*)
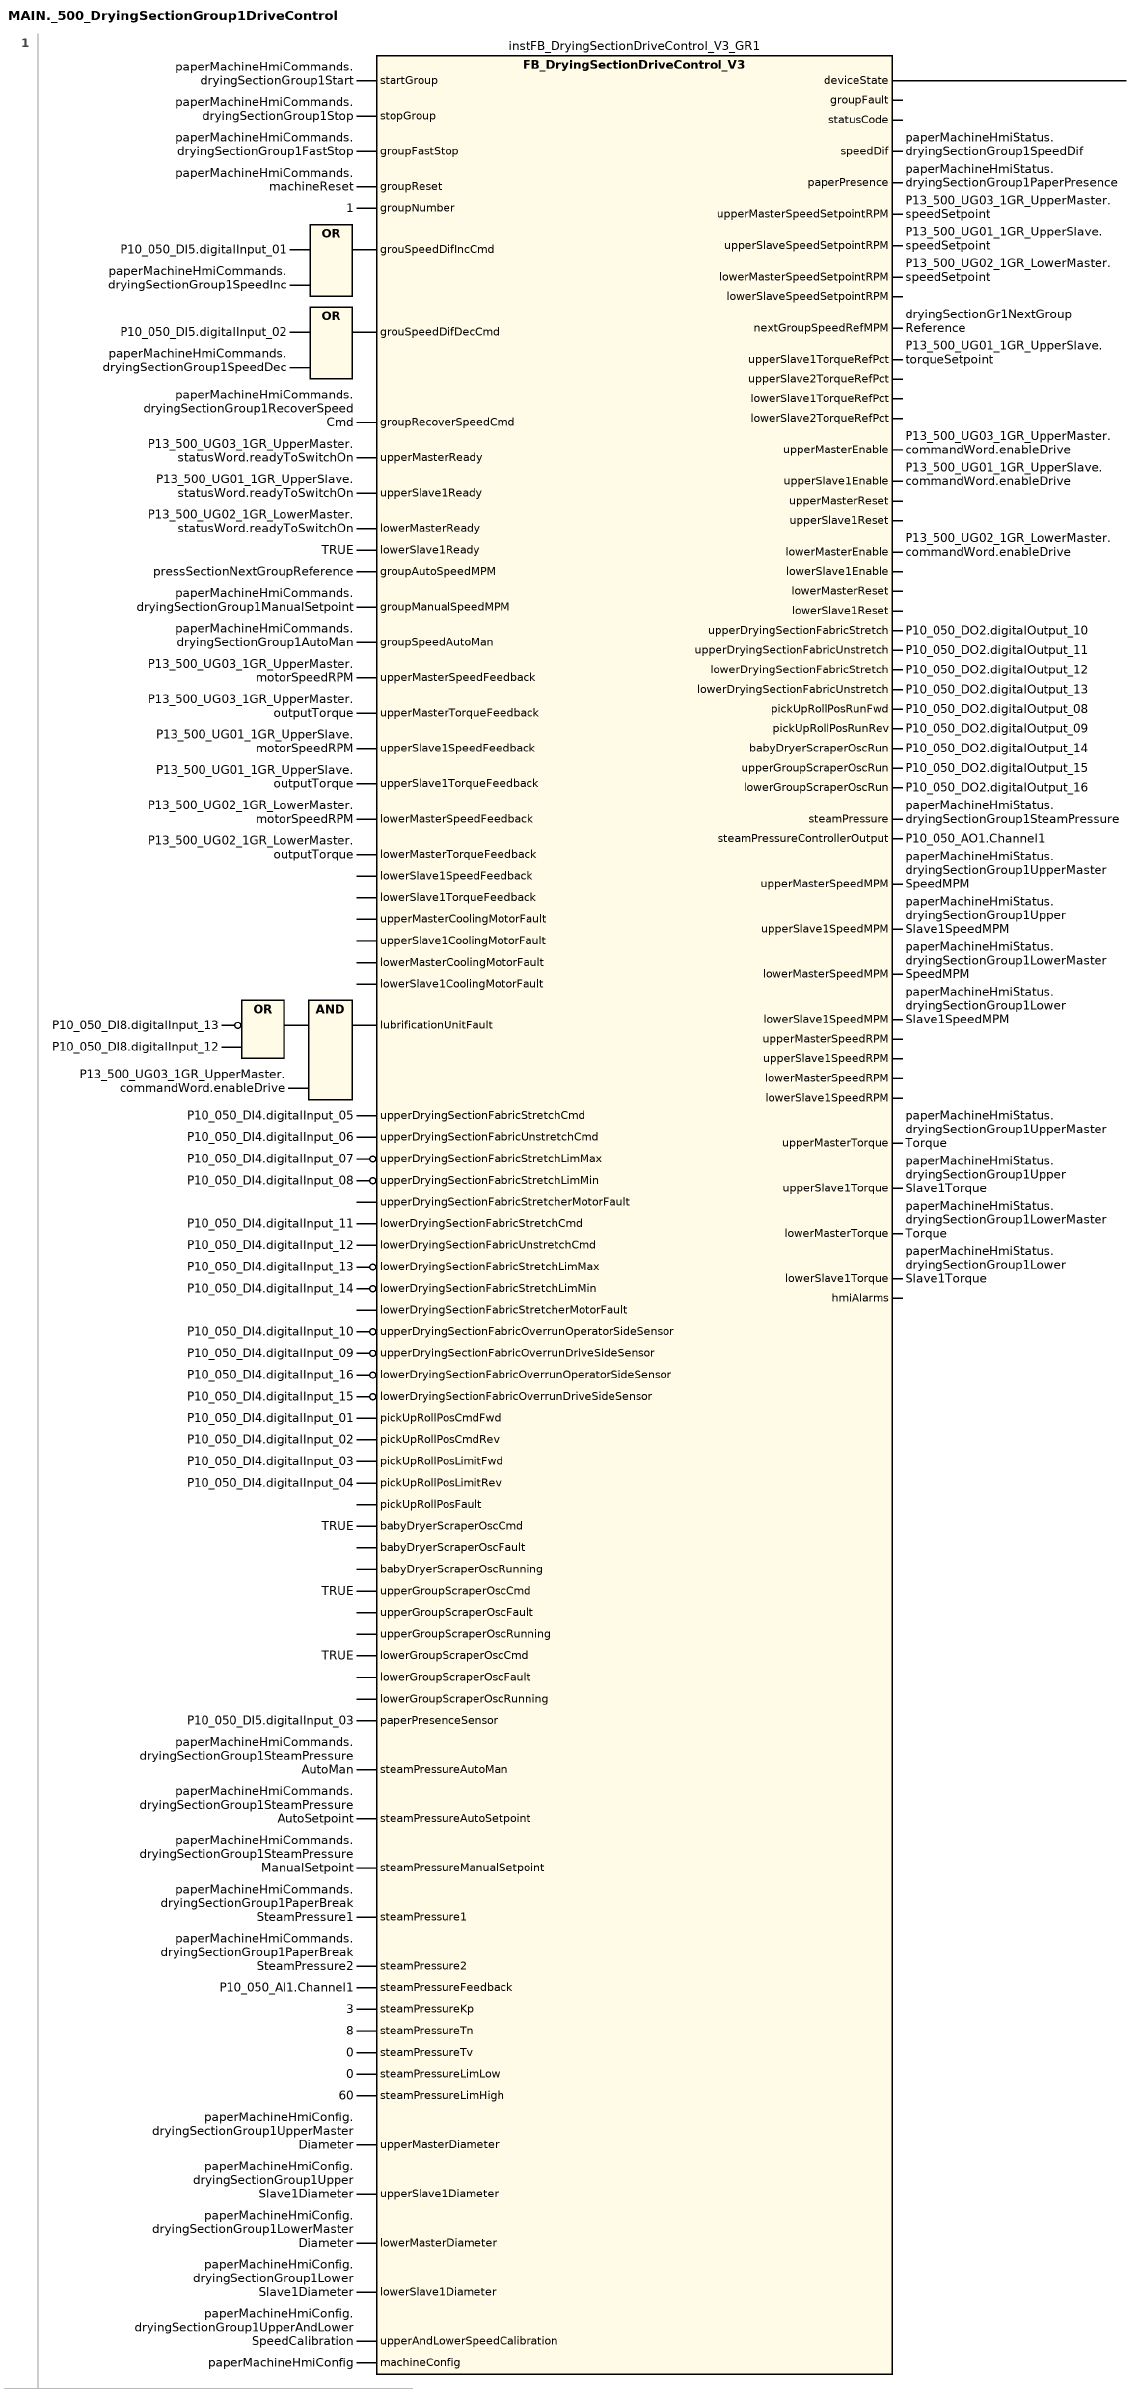
// NETWORK 1
instFB_DryingSectionDriveControl_V3_GR1(
    startGroup := paperMachineHmiCommands.dryingSectionGroup1Start,
    stopGroup := paperMachineHmiCommands.dryingSectionGroup1Stop,
    groupFastStop := paperMachineHmiCommands.dryingSectionGroup1FastStop,
    groupReset := paperMachineHmiCommands.machineReset,
    groupNumber := 1,
    grouSpeedDifIncCmd := P10_050_DI5.digitalInput_01 OR paperMachineHmiCommands.dryingSectionGroup1SpeedInc,
    grouSpeedDifDecCmd := P10_050_DI5.digitalInput_02 OR paperMachineHmiCommands.dryingSectionGroup1SpeedDec,
    groupRecoverSpeedCmd := paperMachineHmiCommands.dryingSectionGroup1RecoverSpeedCmd,
    upperMasterReady := P13_500_UG03_1GR_UpperMaster.statusWord.readyToSwitchOn,
    upperSlave1Ready := P13_500_UG01_1GR_UpperSlave.statusWord.readyToSwitchOn,
    lowerMasterReady := P13_500_UG02_1GR_LowerMaster.statusWord.readyToSwitchOn,
    lowerSlave1Ready := TRUE,
    groupAutoSpeedMPM := pressSectionNextGroupReference,
    groupManualSpeedMPM := paperMachineHmiCommands.dryingSectionGroup1ManualSetpoint,
    groupSpeedAutoMan := paperMachineHmiCommands.dryingSectionGroup1AutoMan,
    upperMasterSpeedFeedback := P13_500_UG03_1GR_UpperMaster.motorSpeedRPM,
    upperMasterTorqueFeedback := P13_500_UG03_1GR_UpperMaster.outputTorque,
    upperSlave1SpeedFeedback := P13_500_UG01_1GR_UpperSlave.motorSpeedRPM,
    upperSlave1TorqueFeedback := P13_500_UG01_1GR_UpperSlave.outputTorque,
    lowerMasterSpeedFeedback := P13_500_UG02_1GR_LowerMaster.motorSpeedRPM,
    lowerMasterTorqueFeedback := P13_500_UG02_1GR_LowerMaster.outputTorque,
    lubrificationUnitFault := (NOT P10_050_DI8.digitalInput_13 OR P10_050_DI8.digitalInput_12) AND P13_500_UG03_1GR_UpperMaster.commandWord.enableDrive,
    upperDryingSectionFabricStretchCmd := P10_050_DI4.digitalInput_05,
    upperDryingSectionFabricUnstretchCmd := P10_050_DI4.digitalInput_06,
    upperDryingSectionFabricStretchLimMax := NOT P10_050_DI4.digitalInput_07,
    upperDryingSectionFabricStretchLimMin := NOT P10_050_DI4.digitalInput_08,
    lowerDryingSectionFabricStretchCmd := P10_050_DI4.digitalInput_11,
    lowerDryingSectionFabricUnstretchCmd := P10_050_DI4.digitalInput_12,
    lowerDryingSectionFabricStretchLimMax := NOT P10_050_DI4.digitalInput_13,
    lowerDryingSectionFabricStretchLimMin := NOT P10_050_DI4.digitalInput_14,
    upperDryingSectionFabricOverrunOperatorSideSensor := NOT P10_050_DI4.digitalInput_10,
    upperDryingSectionFabricOverrunDriveSideSensor := NOT P10_050_DI4.digitalInput_09,
    lowerDryingSectionFabricOverrunOperatorSideSensor := NOT P10_050_DI4.digitalInput_16,
    lowerDryingSectionFabricOverrunDriveSideSensor := NOT P10_050_DI4.digitalInput_15,
    pickUpRollPosCmdFwd := P10_050_DI4.digitalInput_01,
    pickUpRollPosCmdRev := P10_050_DI4.digitalInput_02,
    pickUpRollPosLimitFwd := P10_050_DI4.digitalInput_03,
    pickUpRollPosLimitRev := P10_050_DI4.digitalInput_04,
    babyDryerScraperOscCmd := TRUE,
    upperGroupScraperOscCmd := TRUE,
    lowerGroupScraperOscCmd := TRUE,
    paperPresenceSensor := P10_050_DI5.digitalInput_03,
    steamPressureAutoMan := paperMachineHmiCommands.dryingSectionGroup1SteamPressureAutoMan,
    steamPressureAutoSetpoint := paperMachineHmiCommands.dryingSectionGroup1SteamPressureAutoSetpoint,
    steamPressureManualSetpoint := paperMachineHmiCommands.dryingSectionGroup1SteamPressureManualSetpoint,
    steamPressure1 := paperMachineHmiCommands.dryingSectionGroup1PaperBreakSteamPressure1,
    steamPressure2 := paperMachineHmiCommands.dryingSectionGroup1PaperBreakSteamPressure2,
    steamPressureFeedback := P10_050_AI1.Channel1,
    steamPressureKp := 3,
    steamPressureTn := 8,
    steamPressureTv := 0,
    steamPressureLimLow := 0,
    steamPressureLimHigh := 60,
    upperMasterDiameter := paperMachineHmiConfig.dryingSectionGroup1UpperMasterDiameter,
    upperSlave1Diameter := paperMachineHmiConfig.dryingSectionGroup1UpperSlave1Diameter,
    lowerMasterDiameter := paperMachineHmiConfig.dryingSectionGroup1LowerMasterDiameter,
    lowerSlave1Diameter := paperMachineHmiConfig.dryingSectionGroup1LowerSlave1Diameter,
    upperAndLowerSpeedCalibration := paperMachineHmiConfig.dryingSectionGroup1UpperAndLowerSpeedCalibration,
    machineConfig := paperMachineHmiConfig,
    speedDif => paperMachineHmiStatus.dryingSectionGroup1SpeedDif,
    paperPresence => paperMachineHmiStatus.dryingSectionGroup1PaperPresence,
    upperMasterSpeedSetpointRPM => P13_500_UG03_1GR_UpperMaster.speedSetpoint,
    upperSlaveSpeedSetpointRPM => P13_500_UG01_1GR_UpperSlave.speedSetpoint,
    lowerMasterSpeedSetpointRPM => P13_500_UG02_1GR_LowerMaster.speedSetpoint,
    nextGroupSpeedRefMPM => dryingSectionGr1NextGroupReference,
    upperSlave1TorqueRefPct => P13_500_UG01_1GR_UpperSlave.torqueSetpoint,
    upperMasterEnable => P13_500_UG03_1GR_UpperMaster.commandWord.enableDrive,
    upperSlave1Enable => P13_500_UG01_1GR_UpperSlave.commandWord.enableDrive,
    lowerMasterEnable => P13_500_UG02_1GR_LowerMaster.commandWord.enableDrive,
    upperDryingSectionFabricStretch => P10_050_DO2.digitalOutput_10,
    upperDryingSectionFabricUnstretch => P10_050_DO2.digitalOutput_11,
    lowerDryingSectionFabricStretch => P10_050_DO2.digitalOutput_12,
    lowerDryingSectionFabricUnstretch => P10_050_DO2.digitalOutput_13,
    pickUpRollPosRunFwd => P10_050_DO2.digitalOutput_08,
    pickUpRollPosRunRev => P10_050_DO2.digitalOutput_09,
    babyDryerScraperOscRun => P10_050_DO2.digitalOutput_14,
    upperGroupScraperOscRun => P10_050_DO2.digitalOutput_15,
    lowerGroupScraperOscRun => P10_050_DO2.digitalOutput_16,
    steamPressure => paperMachineHmiStatus.dryingSectionGroup1SteamPressure,
    steamPressureControllerOutput => P10_050_AO1.Channel1,
    upperMasterSpeedMPM => paperMachineHmiStatus.dryingSectionGroup1UpperMasterSpeedMPM,
    upperSlave1SpeedMPM => paperMachineHmiStatus.dryingSectionGroup1UpperSlave1SpeedMPM,
    lowerMasterSpeedMPM => paperMachineHmiStatus.dryingSectionGroup1LowerMasterSpeedMPM,
    lowerSlave1SpeedMPM => paperMachineHmiStatus.dryingSectionGroup1LowerSlave1SpeedMPM,
    upperMasterTorque => paperMachineHmiStatus.dryingSectionGroup1UpperMasterTorque,
    upperSlave1Torque => paperMachineHmiStatus.dryingSectionGroup1UpperSlave1Torque,
    lowerMasterTorque => paperMachineHmiStatus.dryingSectionGroup1LowerMasterTorque,
    lowerSlave1Torque => paperMachineHmiStatus.dryingSectionGroup1LowerSlave1Torque); // FB_DryingSectionDriveControl_V3
END_METHOD

METHOD _501_DryingSectionGroup2DriveControl
VAR_INPUT
END_VAR
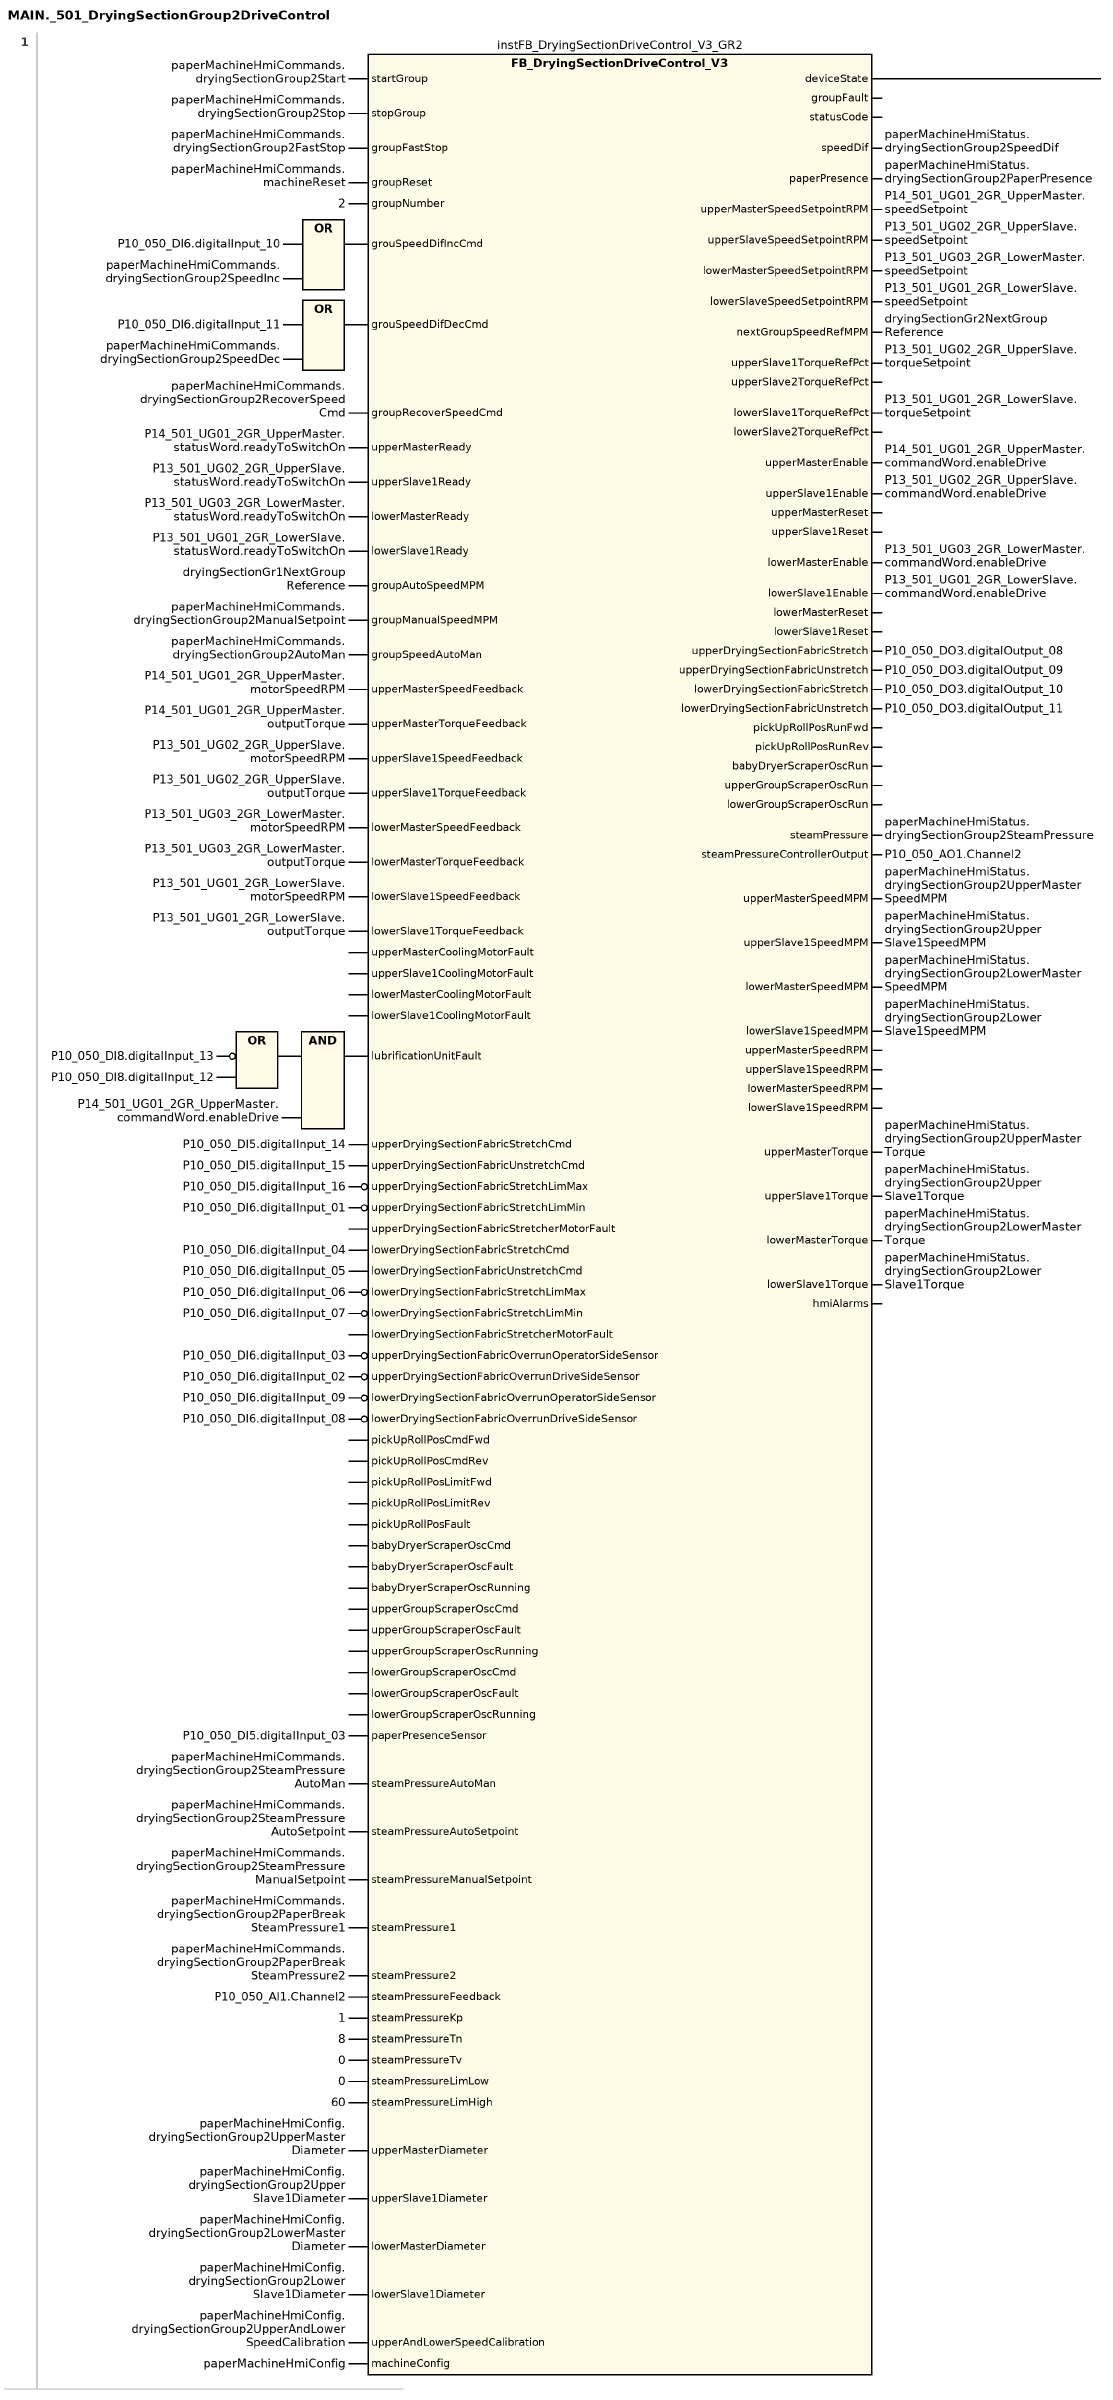
// NETWORK 1
instFB_DryingSectionDriveControl_V3_GR2(
    startGroup := paperMachineHmiCommands.dryingSectionGroup2Start,
    stopGroup := paperMachineHmiCommands.dryingSectionGroup2Stop,
    groupFastStop := paperMachineHmiCommands.dryingSectionGroup2FastStop,
    groupReset := paperMachineHmiCommands.machineReset,
    groupNumber := 2,
    grouSpeedDifIncCmd := P10_050_DI6.digitalInput_10 OR paperMachineHmiCommands.dryingSectionGroup2SpeedInc,
    grouSpeedDifDecCmd := P10_050_DI6.digitalInput_11 OR paperMachineHmiCommands.dryingSectionGroup2SpeedDec,
    groupRecoverSpeedCmd := paperMachineHmiCommands.dryingSectionGroup2RecoverSpeedCmd,
    upperMasterReady := P14_501_UG01_2GR_UpperMaster.statusWord.readyToSwitchOn,
    upperSlave1Ready := P13_501_UG02_2GR_UpperSlave.statusWord.readyToSwitchOn,
    lowerMasterReady := P13_501_UG03_2GR_LowerMaster.statusWord.readyToSwitchOn,
    lowerSlave1Ready := P13_501_UG01_2GR_LowerSlave.statusWord.readyToSwitchOn,
    groupAutoSpeedMPM := dryingSectionGr1NextGroupReference,
    groupManualSpeedMPM := paperMachineHmiCommands.dryingSectionGroup2ManualSetpoint,
    groupSpeedAutoMan := paperMachineHmiCommands.dryingSectionGroup2AutoMan,
    upperMasterSpeedFeedback := P14_501_UG01_2GR_UpperMaster.motorSpeedRPM,
    upperMasterTorqueFeedback := P14_501_UG01_2GR_UpperMaster.outputTorque,
    upperSlave1SpeedFeedback := P13_501_UG02_2GR_UpperSlave.motorSpeedRPM,
    upperSlave1TorqueFeedback := P13_501_UG02_2GR_UpperSlave.outputTorque,
    lowerMasterSpeedFeedback := P13_501_UG03_2GR_LowerMaster.motorSpeedRPM,
    lowerMasterTorqueFeedback := P13_501_UG03_2GR_LowerMaster.outputTorque,
    lowerSlave1SpeedFeedback := P13_501_UG01_2GR_LowerSlave.motorSpeedRPM,
    lowerSlave1TorqueFeedback := P13_501_UG01_2GR_LowerSlave.outputTorque,
    lubrificationUnitFault := (NOT P10_050_DI8.digitalInput_13 OR P10_050_DI8.digitalInput_12) AND P14_501_UG01_2GR_UpperMaster.commandWord.enableDrive,
    upperDryingSectionFabricStretchCmd := P10_050_DI5.digitalInput_14,
    upperDryingSectionFabricUnstretchCmd := P10_050_DI5.digitalInput_15,
    upperDryingSectionFabricStretchLimMax := NOT P10_050_DI5.digitalInput_16,
    upperDryingSectionFabricStretchLimMin := NOT P10_050_DI6.digitalInput_01,
    lowerDryingSectionFabricStretchCmd := P10_050_DI6.digitalInput_04,
    lowerDryingSectionFabricUnstretchCmd := P10_050_DI6.digitalInput_05,
    lowerDryingSectionFabricStretchLimMax := NOT P10_050_DI6.digitalInput_06,
    lowerDryingSectionFabricStretchLimMin := NOT P10_050_DI6.digitalInput_07,
    upperDryingSectionFabricOverrunOperatorSideSensor := NOT P10_050_DI6.digitalInput_03,
    upperDryingSectionFabricOverrunDriveSideSensor := NOT P10_050_DI6.digitalInput_02,
    lowerDryingSectionFabricOverrunOperatorSideSensor := NOT P10_050_DI6.digitalInput_09,
    lowerDryingSectionFabricOverrunDriveSideSensor := NOT P10_050_DI6.digitalInput_08,
    paperPresenceSensor := P10_050_DI5.digitalInput_03,
    steamPressureAutoMan := paperMachineHmiCommands.dryingSectionGroup2SteamPressureAutoMan,
    steamPressureAutoSetpoint := paperMachineHmiCommands.dryingSectionGroup2SteamPressureAutoSetpoint,
    steamPressureManualSetpoint := paperMachineHmiCommands.dryingSectionGroup2SteamPressureManualSetpoint,
    steamPressure1 := paperMachineHmiCommands.dryingSectionGroup2PaperBreakSteamPressure1,
    steamPressure2 := paperMachineHmiCommands.dryingSectionGroup2PaperBreakSteamPressure2,
    steamPressureFeedback := P10_050_AI1.Channel2,
    steamPressureKp := 1,
    steamPressureTn := 8,
    steamPressureTv := 0,
    steamPressureLimLow := 0,
    steamPressureLimHigh := 60,
    upperMasterDiameter := paperMachineHmiConfig.dryingSectionGroup2UpperMasterDiameter,
    upperSlave1Diameter := paperMachineHmiConfig.dryingSectionGroup2UpperSlave1Diameter,
    lowerMasterDiameter := paperMachineHmiConfig.dryingSectionGroup2LowerMasterDiameter,
    lowerSlave1Diameter := paperMachineHmiConfig.dryingSectionGroup2LowerSlave1Diameter,
    upperAndLowerSpeedCalibration := paperMachineHmiConfig.dryingSectionGroup2UpperAndLowerSpeedCalibration,
    machineConfig := paperMachineHmiConfig,
    speedDif => paperMachineHmiStatus.dryingSectionGroup2SpeedDif,
    paperPresence => paperMachineHmiStatus.dryingSectionGroup2PaperPresence,
    upperMasterSpeedSetpointRPM => P14_501_UG01_2GR_UpperMaster.speedSetpoint,
    upperSlaveSpeedSetpointRPM => P13_501_UG02_2GR_UpperSlave.speedSetpoint,
    lowerMasterSpeedSetpointRPM => P13_501_UG03_2GR_LowerMaster.speedSetpoint,
    lowerSlaveSpeedSetpointRPM => P13_501_UG01_2GR_LowerSlave.speedSetpoint,
    nextGroupSpeedRefMPM => dryingSectionGr2NextGroupReference,
    upperSlave1TorqueRefPct => P13_501_UG02_2GR_UpperSlave.torqueSetpoint,
    lowerSlave1TorqueRefPct => P13_501_UG01_2GR_LowerSlave.torqueSetpoint,
    upperMasterEnable => P14_501_UG01_2GR_UpperMaster.commandWord.enableDrive,
    upperSlave1Enable => P13_501_UG02_2GR_UpperSlave.commandWord.enableDrive,
    lowerMasterEnable => P13_501_UG03_2GR_LowerMaster.commandWord.enableDrive,
    lowerSlave1Enable => P13_501_UG01_2GR_LowerSlave.commandWord.enableDrive,
    upperDryingSectionFabricStretch => P10_050_DO3.digitalOutput_08,
    upperDryingSectionFabricUnstretch => P10_050_DO3.digitalOutput_09,
    lowerDryingSectionFabricStretch => P10_050_DO3.digitalOutput_10,
    lowerDryingSectionFabricUnstretch => P10_050_DO3.digitalOutput_11,
    steamPressure => paperMachineHmiStatus.dryingSectionGroup2SteamPressure,
    steamPressureControllerOutput => P10_050_AO1.Channel2,
    upperMasterSpeedMPM => paperMachineHmiStatus.dryingSectionGroup2UpperMasterSpeedMPM,
    upperSlave1SpeedMPM => paperMachineHmiStatus.dryingSectionGroup2UpperSlave1SpeedMPM,
    lowerMasterSpeedMPM => paperMachineHmiStatus.dryingSectionGroup2LowerMasterSpeedMPM,
    lowerSlave1SpeedMPM => paperMachineHmiStatus.dryingSectionGroup2LowerSlave1SpeedMPM,
    upperMasterTorque => paperMachineHmiStatus.dryingSectionGroup2UpperMasterTorque,
    upperSlave1Torque => paperMachineHmiStatus.dryingSectionGroup2UpperSlave1Torque,
    lowerMasterTorque => paperMachineHmiStatus.dryingSectionGroup2LowerMasterTorque,
    lowerSlave1Torque => paperMachineHmiStatus.dryingSectionGroup2LowerSlave1Torque); // FB_DryingSectionDriveControl_V3
END_METHOD

METHOD _502_DryingSectionGroup3DriveControl
VAR_INPUT
END_VAR
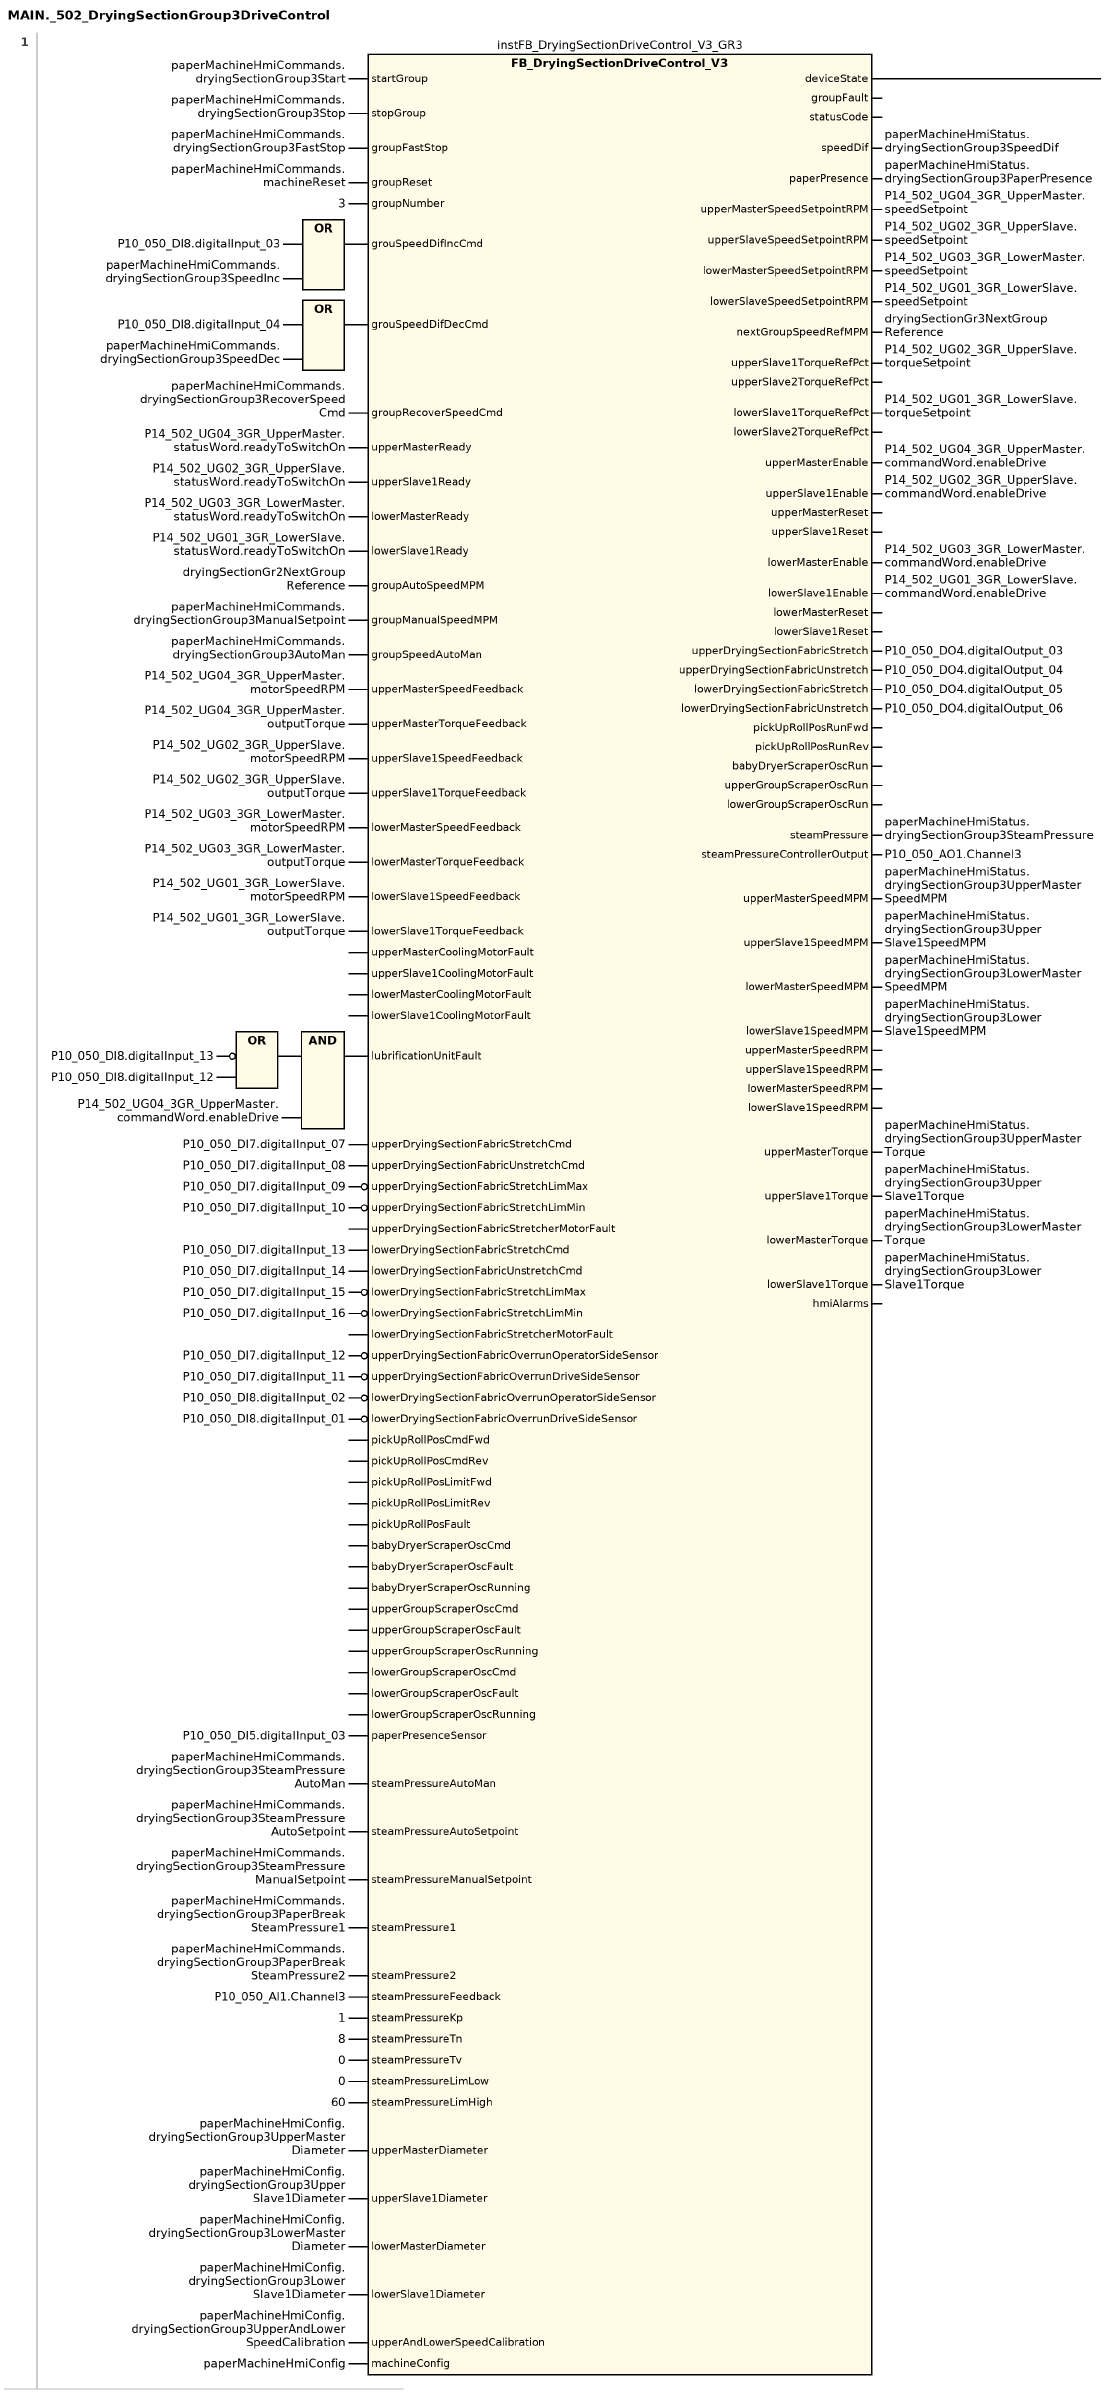
// NETWORK 1
instFB_DryingSectionDriveControl_V3_GR3(
    startGroup := paperMachineHmiCommands.dryingSectionGroup3Start,
    stopGroup := paperMachineHmiCommands.dryingSectionGroup3Stop,
    groupFastStop := paperMachineHmiCommands.dryingSectionGroup3FastStop,
    groupReset := paperMachineHmiCommands.machineReset,
    groupNumber := 3,
    grouSpeedDifIncCmd := P10_050_DI8.digitalInput_03 OR paperMachineHmiCommands.dryingSectionGroup3SpeedInc,
    grouSpeedDifDecCmd := P10_050_DI8.digitalInput_04 OR paperMachineHmiCommands.dryingSectionGroup3SpeedDec,
    groupRecoverSpeedCmd := paperMachineHmiCommands.dryingSectionGroup3RecoverSpeedCmd,
    upperMasterReady := P14_502_UG04_3GR_UpperMaster.statusWord.readyToSwitchOn,
    upperSlave1Ready := P14_502_UG02_3GR_UpperSlave.statusWord.readyToSwitchOn,
    lowerMasterReady := P14_502_UG03_3GR_LowerMaster.statusWord.readyToSwitchOn,
    lowerSlave1Ready := P14_502_UG01_3GR_LowerSlave.statusWord.readyToSwitchOn,
    groupAutoSpeedMPM := dryingSectionGr2NextGroupReference,
    groupManualSpeedMPM := paperMachineHmiCommands.dryingSectionGroup3ManualSetpoint,
    groupSpeedAutoMan := paperMachineHmiCommands.dryingSectionGroup3AutoMan,
    upperMasterSpeedFeedback := P14_502_UG04_3GR_UpperMaster.motorSpeedRPM,
    upperMasterTorqueFeedback := P14_502_UG04_3GR_UpperMaster.outputTorque,
    upperSlave1SpeedFeedback := P14_502_UG02_3GR_UpperSlave.motorSpeedRPM,
    upperSlave1TorqueFeedback := P14_502_UG02_3GR_UpperSlave.outputTorque,
    lowerMasterSpeedFeedback := P14_502_UG03_3GR_LowerMaster.motorSpeedRPM,
    lowerMasterTorqueFeedback := P14_502_UG03_3GR_LowerMaster.outputTorque,
    lowerSlave1SpeedFeedback := P14_502_UG01_3GR_LowerSlave.motorSpeedRPM,
    lowerSlave1TorqueFeedback := P14_502_UG01_3GR_LowerSlave.outputTorque,
    lubrificationUnitFault := (NOT P10_050_DI8.digitalInput_13 OR P10_050_DI8.digitalInput_12) AND P14_502_UG04_3GR_UpperMaster.commandWord.enableDrive,
    upperDryingSectionFabricStretchCmd := P10_050_DI7.digitalInput_07,
    upperDryingSectionFabricUnstretchCmd := P10_050_DI7.digitalInput_08,
    upperDryingSectionFabricStretchLimMax := NOT P10_050_DI7.digitalInput_09,
    upperDryingSectionFabricStretchLimMin := NOT P10_050_DI7.digitalInput_10,
    lowerDryingSectionFabricStretchCmd := P10_050_DI7.digitalInput_13,
    lowerDryingSectionFabricUnstretchCmd := P10_050_DI7.digitalInput_14,
    lowerDryingSectionFabricStretchLimMax := NOT P10_050_DI7.digitalInput_15,
    lowerDryingSectionFabricStretchLimMin := NOT P10_050_DI7.digitalInput_16,
    upperDryingSectionFabricOverrunOperatorSideSensor := NOT P10_050_DI7.digitalInput_12,
    upperDryingSectionFabricOverrunDriveSideSensor := NOT P10_050_DI7.digitalInput_11,
    lowerDryingSectionFabricOverrunOperatorSideSensor := NOT P10_050_DI8.digitalInput_02,
    lowerDryingSectionFabricOverrunDriveSideSensor := NOT P10_050_DI8.digitalInput_01,
    paperPresenceSensor := P10_050_DI5.digitalInput_03,
    steamPressureAutoMan := paperMachineHmiCommands.dryingSectionGroup3SteamPressureAutoMan,
    steamPressureAutoSetpoint := paperMachineHmiCommands.dryingSectionGroup3SteamPressureAutoSetpoint,
    steamPressureManualSetpoint := paperMachineHmiCommands.dryingSectionGroup3SteamPressureManualSetpoint,
    steamPressure1 := paperMachineHmiCommands.dryingSectionGroup3PaperBreakSteamPressure1,
    steamPressure2 := paperMachineHmiCommands.dryingSectionGroup3PaperBreakSteamPressure2,
    steamPressureFeedback := P10_050_AI1.Channel3,
    steamPressureKp := 1,
    steamPressureTn := 8,
    steamPressureTv := 0,
    steamPressureLimLow := 0,
    steamPressureLimHigh := 60,
    upperMasterDiameter := paperMachineHmiConfig.dryingSectionGroup3UpperMasterDiameter,
    upperSlave1Diameter := paperMachineHmiConfig.dryingSectionGroup3UpperSlave1Diameter,
    lowerMasterDiameter := paperMachineHmiConfig.dryingSectionGroup3LowerMasterDiameter,
    lowerSlave1Diameter := paperMachineHmiConfig.dryingSectionGroup3LowerSlave1Diameter,
    upperAndLowerSpeedCalibration := paperMachineHmiConfig.dryingSectionGroup3UpperAndLowerSpeedCalibration,
    machineConfig := paperMachineHmiConfig,
    speedDif => paperMachineHmiStatus.dryingSectionGroup3SpeedDif,
    paperPresence => paperMachineHmiStatus.dryingSectionGroup3PaperPresence,
    upperMasterSpeedSetpointRPM => P14_502_UG04_3GR_UpperMaster.speedSetpoint,
    upperSlaveSpeedSetpointRPM => P14_502_UG02_3GR_UpperSlave.speedSetpoint,
    lowerMasterSpeedSetpointRPM => P14_502_UG03_3GR_LowerMaster.speedSetpoint,
    lowerSlaveSpeedSetpointRPM => P14_502_UG01_3GR_LowerSlave.speedSetpoint,
    nextGroupSpeedRefMPM => dryingSectionGr3NextGroupReference,
    upperSlave1TorqueRefPct => P14_502_UG02_3GR_UpperSlave.torqueSetpoint,
    lowerSlave1TorqueRefPct => P14_502_UG01_3GR_LowerSlave.torqueSetpoint,
    upperMasterEnable => P14_502_UG04_3GR_UpperMaster.commandWord.enableDrive,
    upperSlave1Enable => P14_502_UG02_3GR_UpperSlave.commandWord.enableDrive,
    lowerMasterEnable => P14_502_UG03_3GR_LowerMaster.commandWord.enableDrive,
    lowerSlave1Enable => P14_502_UG01_3GR_LowerSlave.commandWord.enableDrive,
    upperDryingSectionFabricStretch => P10_050_DO4.digitalOutput_03,
    upperDryingSectionFabricUnstretch => P10_050_DO4.digitalOutput_04,
    lowerDryingSectionFabricStretch => P10_050_DO4.digitalOutput_05,
    lowerDryingSectionFabricUnstretch => P10_050_DO4.digitalOutput_06,
    steamPressure => paperMachineHmiStatus.dryingSectionGroup3SteamPressure,
    steamPressureControllerOutput => P10_050_AO1.Channel3,
    upperMasterSpeedMPM => paperMachineHmiStatus.dryingSectionGroup3UpperMasterSpeedMPM,
    upperSlave1SpeedMPM => paperMachineHmiStatus.dryingSectionGroup3UpperSlave1SpeedMPM,
    lowerMasterSpeedMPM => paperMachineHmiStatus.dryingSectionGroup3LowerMasterSpeedMPM,
    lowerSlave1SpeedMPM => paperMachineHmiStatus.dryingSectionGroup3LowerSlave1SpeedMPM,
    upperMasterTorque => paperMachineHmiStatus.dryingSectionGroup3UpperMasterTorque,
    upperSlave1Torque => paperMachineHmiStatus.dryingSectionGroup3UpperSlave1Torque,
    lowerMasterTorque => paperMachineHmiStatus.dryingSectionGroup3LowerMasterTorque,
    lowerSlave1Torque => paperMachineHmiStatus.dryingSectionGroup3LowerSlave1Torque); // FB_DryingSectionDriveControl_V3
END_METHOD

METHOD _550_DryingSectionLubrification
VAR_INPUT
END_VAR
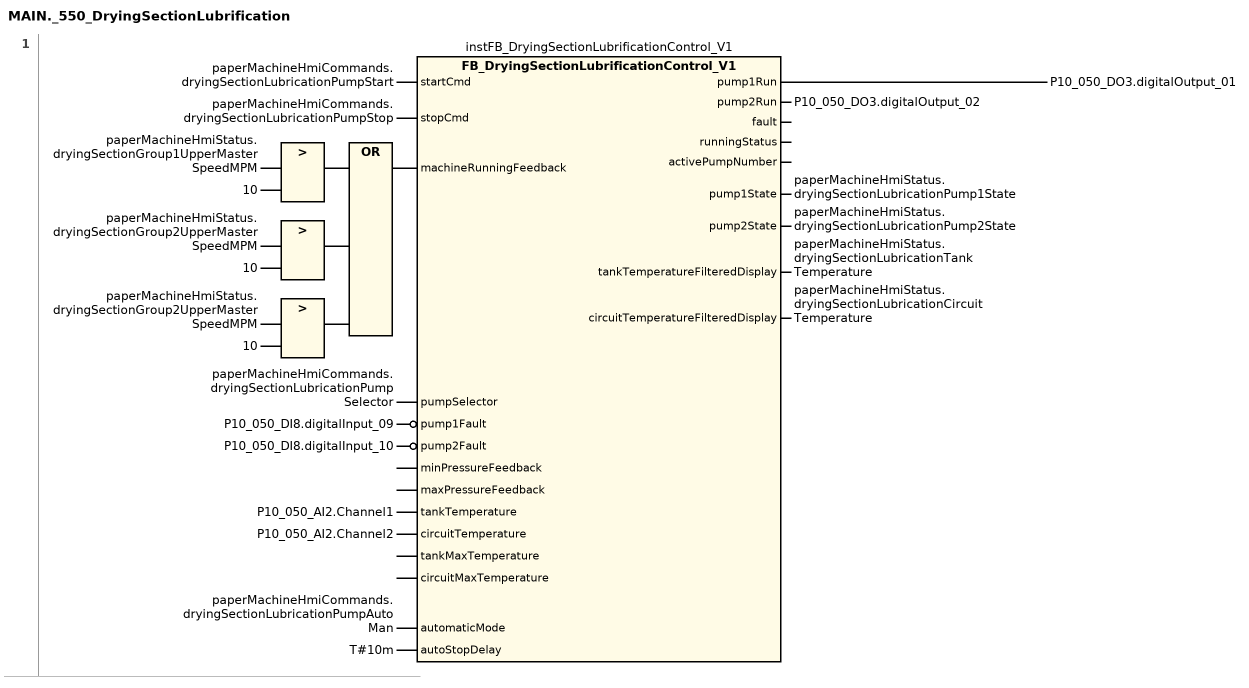
// NETWORK 1
instFB_DryingSectionLubrificationControl_V1(
    startCmd := paperMachineHmiCommands.dryingSectionLubricationPumpStart,
    stopCmd := paperMachineHmiCommands.dryingSectionLubricationPumpStop,
    machineRunningFeedback := paperMachineHmiStatus.dryingSectionGroup1UpperMasterSpeedMPM > 10 OR paperMachineHmiStatus.dryingSectionGroup2UpperMasterSpeedMPM > 10 OR paperMachineHmiStatus.dryingSectionGroup2UpperMasterSpeedMPM > 10,
    pumpSelector := paperMachineHmiCommands.dryingSectionLubricationPumpSelector,
    pump1Fault := NOT P10_050_DI8.digitalInput_09,
    pump2Fault := NOT P10_050_DI8.digitalInput_10,
    tankTemperature := P10_050_AI2.Channel1,
    circuitTemperature := P10_050_AI2.Channel2,
    automaticMode := paperMachineHmiCommands.dryingSectionLubricationPumpAutoMan,
    autoStopDelay := T#10m,
    pump2Run => P10_050_DO3.digitalOutput_02,
    pump1State => paperMachineHmiStatus.dryingSectionLubricationPump1State,
    pump2State => paperMachineHmiStatus.dryingSectionLubricationPump2State,
    tankTemperatureFilteredDisplay => paperMachineHmiStatus.dryingSectionLubricationTankTemperature,
    circuitTemperatureFilteredDisplay => paperMachineHmiStatus.dryingSectionLubricationCircuitTemperature); // FB_DryingSectionLubrificationControl_V1
P10_050_DO3.digitalOutput_01 := instFB_DryingSectionLubrificationControl_V1.pump1Run;
END_METHOD

METHOD _600_WinderGroup
VAR_INPUT
END_VAR
(*
	winderPressureSetpointOperatorSide : REAL; // EN: Controller output (operator side) / PT: Saída do controlador (lado operador)
    winderPressureSetpointDriveSide    : REAL; // EN: Controller output (drive side) / PT: Saída do controlador (lado motriz)
	winderSpeedMPM   : REAL;  // Group 2 Upper Slave 2 speed [m/min or rpm] (Velocidade do motor escravo 2 superior do grupo 2)
	winderTorque  : REAL;  // Group 2 Upper Slave 2 torque [% or Nm] (Torque do motor escravo 2 superior do grupo 2)
	winderState   : INT;   // Group 2 Upper Slave 2 state code (Estado do motor escravo 2 superior do grupo 2)
*)

(*
	// ─────────────── WINDER SECTION ───────────────
	// Start/stop and speed control commands for the winder section.
	winderSectionStart            : BOOL;  // Start Press Section (Ligar Prensa)
	winderSectionStop             : BOOL;  // Stop Press Section (Parar Prensa)
	winderSectionAutoMan          : BOOL;  // 1 = Auto / 0 = Manual mode (Modo automático/manual)
	winderSectionManualSetpoint   : REAL;  // Manual speed setpoint [m/min] (Setpoint manual)
	winderSectionSpeedInc         : BOOL;  // Increase speed manually (Aumentar velocidade)
	winderSectionSpeedDec         : BOOL;  // Decrease speed manually (Diminuir velocidade)
	winderSectionRecoverSpeedCmd  : BOOL;  // Temporarily recover speed (Recuperar velocidade)
	winderSectionRecoverIncrement : REAL;  // Recovery speed increment [m/min or %] (Incremento de recuperação)


  // Pressure fine adjustments for rider roll
    winderPressureOperatorSideIncCmd : BOOL; // EN: Increase operator-side pressure / PT: Aumenta a pressão no lado do operador
    winderPressureOperatorSideDecCmd : BOOL; // EN: Decrease operator-side pressure / PT: Diminui a pressão no lado do operador

    winderPressureDriveSideIncCmd    : BOOL; // EN: Increase drive-side pressure / PT: Aumenta a pressão no lado motriz
    winderPressureDriveSideDecCmd    : BOOL; // EN: Decrease drive-side pressure / PT: Diminui a pressão no lado motriz

	winderRiderRollWorkPositionCmd	: BOOL;
	winderRiderRollReleasePositionCmd	: BOOL;
	
    //==============================================================
    // CORE LOCK (CHUCK LOCKING SYSTEM)
    //==============================================================
    winderCoreLockAutoMan         : BOOL;  // EN: Core lock mode (0=Manual, 1=Auto) / PT: Modo do travamento do mandril (0=Manual, 1=Automático)
    winderCoreLockCmd             : BOOL;  // EN: Lock core chucks / PT: Travar mandril (core chucks)
    winderCoreUnlockCmd           : BOOL;  // EN: Unlock core chucks / PT: Destravar mandril

	//==============================================================
    // CORE LOCK (CHUCK LOCKING SYSTEM)
    //==============================================================
	winderCoreAceleratorEngageCmd : BOOL;
	winderCoreAceleratorDisengageCmd : BOOL;
	
    //==============================================================
    // CORE BRAKE CONTROL
    //==============================================================
    winderCoreBrakeAutoMan        : BOOL;  // EN: Core brake mode (0=Manual, 1=Auto) / PT: Modo de freio do mandril (0=Manual, 1=Automático)
    winderCoreBrakeEnableCmd      : BOOL;  // EN: Enable core brake / PT: Habilita o freio do mandril
    winderCoreBrakeDisableCmd     : BOOL;  // EN: Disable core brake / PT: Desabilita o freio do mandril	
	
	// ─────────────── WINDER SECTION ───────────────
	// Start/stop and speed control commands for the winder section.
	winderSectionStart            : BOOL;  // Start Press Section (Ligar Prensa)
	winderSectionStop             : BOOL;  // Stop Press Section (Parar Prensa)
	winderSectionAutoMan          : BOOL;  // 1 = Auto / 0 = Manual mode (Modo automático/manual)
	winderSectionManualSetpoint   : REAL;  // Manual speed setpoint [m/min] (Setpoint manual)
	winderSectionSpeedInc         : BOOL;  // Increase speed manually (Aumentar velocidade)
	winderSectionSpeedDec         : BOOL;  // Decrease speed manually (Diminuir velocidade)
	winderSectionRecoverSpeedCmd  : BOOL;  // Temporarily recover speed (Recuperar velocidade)
	winderSectionRecoverIncrement : REAL;  // Recovery speed increment [m/min or %] (Incremento de recuperação)
	
    //==============================================================
    // CORE BRAKE CONTROL
    //==============================================================
    winderCoreBrakeAutoMan        : BOOL;  // EN: Core brake mode (0=Manual, 1=Auto) / PT: Modo de freio do mandril (0=Manual, 1=Automático)
    winderCoreBrakeEnableCmd      : BOOL;  // EN: Enable core brake / PT: Habilita o freio do mandril
    winderCoreBrakeDisableCmd     : BOOL;  // EN: Disable core brake / PT: Desabilita o freio do mandril	
	
	winderCorePositioningArmFwdCmd      : BOOL;  // EN: Command to move arm forward / PT: Comando para avançar o braço posicionador
    winderCorePositioningArmRevCmd      : BOOL;  // EN: Command to move arm backward / PT: Comando para recuar o braço posicionador

    winderCorePositioningArmPosLimitFwd : BOOL;  // EN: Forward limit switch / PT: Fim de curso avançado
    winderCorePositioningArmPosLimitRev : BOOL;  // EN: Reverse limit switch / PT: Fim de curso recuado	
	
	winderEnableTorqueControl			: REAL;

	winderTorqueSetpoint			: REAL;	
	
	
*)

VAR
	winderTorqueSetpoint: REAL;
END_VAR
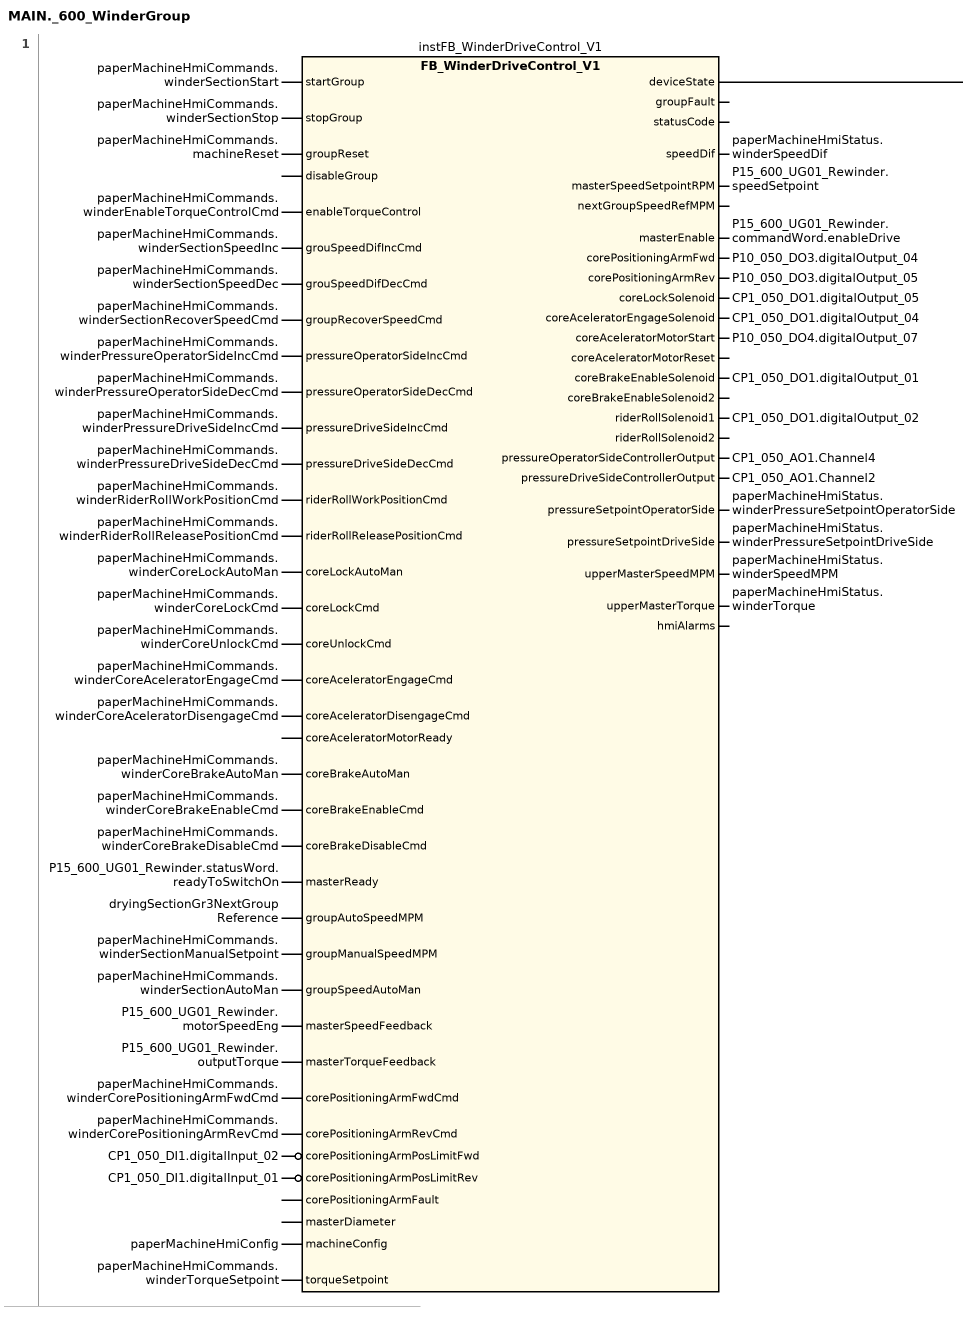
// NETWORK 1
instFB_WinderDriveControl_V1(
    startGroup := paperMachineHmiCommands.winderSectionStart,
    stopGroup := paperMachineHmiCommands.winderSectionStop,
    groupReset := paperMachineHmiCommands.machineReset,
    enableTorqueControl := paperMachineHmiCommands.winderEnableTorqueControlCmd,
    grouSpeedDifIncCmd := paperMachineHmiCommands.winderSectionSpeedInc,
    grouSpeedDifDecCmd := paperMachineHmiCommands.winderSectionSpeedDec,
    groupRecoverSpeedCmd := paperMachineHmiCommands.winderSectionRecoverSpeedCmd,
    pressureOperatorSideIncCmd := paperMachineHmiCommands.winderPressureOperatorSideIncCmd,
    pressureOperatorSideDecCmd := paperMachineHmiCommands.winderPressureOperatorSideDecCmd,
    pressureDriveSideIncCmd := paperMachineHmiCommands.winderPressureDriveSideIncCmd,
    pressureDriveSideDecCmd := paperMachineHmiCommands.winderPressureDriveSideDecCmd,
    riderRollWorkPositionCmd := paperMachineHmiCommands.winderRiderRollWorkPositionCmd,
    riderRollReleasePositionCmd := paperMachineHmiCommands.winderRiderRollReleasePositionCmd,
    coreLockAutoMan := paperMachineHmiCommands.winderCoreLockAutoMan,
    coreLockCmd := paperMachineHmiCommands.winderCoreLockCmd,
    coreUnlockCmd := paperMachineHmiCommands.winderCoreUnlockCmd,
    coreAceleratorEngageCmd := paperMachineHmiCommands.winderCoreAceleratorEngageCmd,
    coreAceleratorDisengageCmd := paperMachineHmiCommands.winderCoreAceleratorDisengageCmd,
    coreBrakeAutoMan := paperMachineHmiCommands.winderCoreBrakeAutoMan,
    coreBrakeEnableCmd := paperMachineHmiCommands.winderCoreBrakeEnableCmd,
    coreBrakeDisableCmd := paperMachineHmiCommands.winderCoreBrakeDisableCmd,
    masterReady := P15_600_UG01_Rewinder.statusWord.readyToSwitchOn,
    groupAutoSpeedMPM := dryingSectionGr3NextGroupReference,
    groupManualSpeedMPM := paperMachineHmiCommands.winderSectionManualSetpoint,
    groupSpeedAutoMan := paperMachineHmiCommands.winderSectionAutoMan,
    masterSpeedFeedback := P15_600_UG01_Rewinder.motorSpeedEng,
    masterTorqueFeedback := P15_600_UG01_Rewinder.outputTorque,
    corePositioningArmFwdCmd := paperMachineHmiCommands.winderCorePositioningArmFwdCmd,
    corePositioningArmRevCmd := paperMachineHmiCommands.winderCorePositioningArmRevCmd,
    corePositioningArmPosLimitFwd := NOT CP1_050_DI1.digitalInput_02,
    corePositioningArmPosLimitRev := NOT CP1_050_DI1.digitalInput_01,
    machineConfig := paperMachineHmiConfig,
    torqueSetpoint := paperMachineHmiCommands.winderTorqueSetpoint,
    speedDif => paperMachineHmiStatus.winderSpeedDif,
    masterSpeedSetpointRPM => P15_600_UG01_Rewinder.speedSetpoint,
    masterEnable => P15_600_UG01_Rewinder.commandWord.enableDrive,
    corePositioningArmFwd => P10_050_DO3.digitalOutput_04,
    corePositioningArmRev => P10_050_DO3.digitalOutput_05,
    coreLockSolenoid => CP1_050_DO1.digitalOutput_05,
    coreAceleratorEngageSolenoid => CP1_050_DO1.digitalOutput_04,
    coreAceleratorMotorStart => P10_050_DO4.digitalOutput_07,
    coreBrakeEnableSolenoid => CP1_050_DO1.digitalOutput_01,
    riderRollSolenoid1 => CP1_050_DO1.digitalOutput_02,
    pressureOperatorSideControllerOutput => CP1_050_AO1.Channel4,
    pressureDriveSideControllerOutput => CP1_050_AO1.Channel2,
    pressureSetpointOperatorSide => paperMachineHmiStatus.winderPressureSetpointOperatorSide,
    pressureSetpointDriveSide => paperMachineHmiStatus.winderPressureSetpointDriveSide,
    upperMasterSpeedMPM => paperMachineHmiStatus.winderSpeedMPM,
    upperMasterTorque => paperMachineHmiStatus.winderTorque); // FB_WinderDriveControl_V1
END_METHOD

METHOD _888_Alarms
VAR_INPUT
END_VAR
(*

FB_AlarmControl
*)
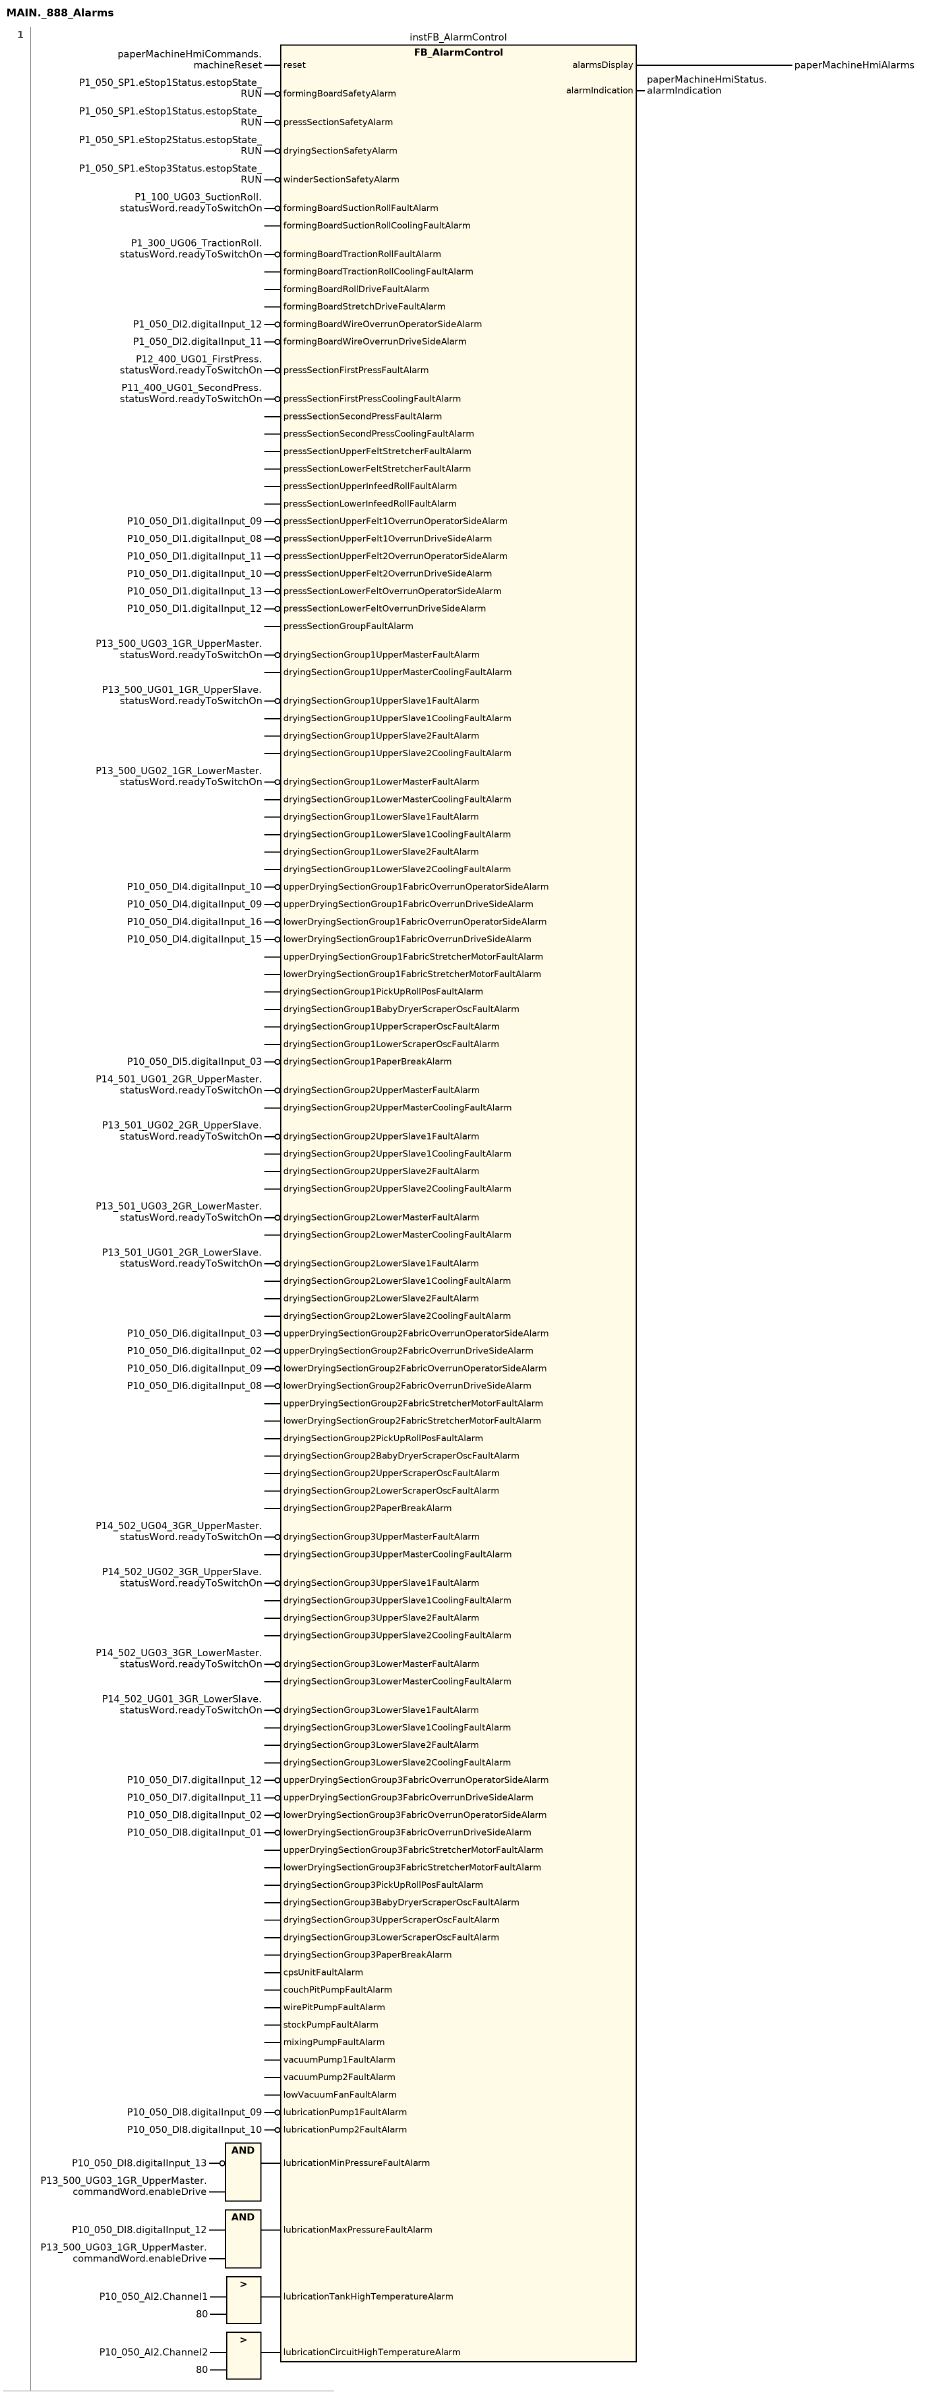
// NETWORK 1
instFB_AlarmControl(
    reset := paperMachineHmiCommands.machineReset,
    formingBoardSafetyAlarm := NOT P1_050_SP1.eStop1Status.estopState_RUN,
    pressSectionSafetyAlarm := NOT P1_050_SP1.eStop1Status.estopState_RUN,
    dryingSectionSafetyAlarm := NOT P1_050_SP1.eStop2Status.estopState_RUN,
    winderSectionSafetyAlarm := NOT P1_050_SP1.eStop3Status.estopState_RUN,
    formingBoardSuctionRollFaultAlarm := NOT P1_100_UG03_SuctionRoll.statusWord.readyToSwitchOn,
    formingBoardTractionRollFaultAlarm := NOT P1_300_UG06_TractionRoll.statusWord.readyToSwitchOn,
    formingBoardWireOverrunOperatorSideAlarm := NOT P1_050_DI2.digitalInput_12,
    formingBoardWireOverrunDriveSideAlarm := NOT P1_050_DI2.digitalInput_11,
    pressSectionFirstPressFaultAlarm := NOT P12_400_UG01_FirstPress.statusWord.readyToSwitchOn,
    pressSectionFirstPressCoolingFaultAlarm := NOT P11_400_UG01_SecondPress.statusWord.readyToSwitchOn,
    pressSectionUpperFelt1OverrunOperatorSideAlarm := NOT P10_050_DI1.digitalInput_09,
    pressSectionUpperFelt1OverrunDriveSideAlarm := NOT P10_050_DI1.digitalInput_08,
    pressSectionUpperFelt2OverrunOperatorSideAlarm := NOT P10_050_DI1.digitalInput_11,
    pressSectionUpperFelt2OverrunDriveSideAlarm := NOT P10_050_DI1.digitalInput_10,
    pressSectionLowerFeltOverrunOperatorSideAlarm := NOT P10_050_DI1.digitalInput_13,
    pressSectionLowerFeltOverrunDriveSideAlarm := NOT P10_050_DI1.digitalInput_12,
    dryingSectionGroup1UpperMasterFaultAlarm := NOT P13_500_UG03_1GR_UpperMaster.statusWord.readyToSwitchOn,
    dryingSectionGroup1UpperSlave1FaultAlarm := NOT P13_500_UG01_1GR_UpperSlave.statusWord.readyToSwitchOn,
    dryingSectionGroup1LowerMasterFaultAlarm := NOT P13_500_UG02_1GR_LowerMaster.statusWord.readyToSwitchOn,
    upperDryingSectionGroup1FabricOverrunOperatorSideAlarm := NOT P10_050_DI4.digitalInput_10,
    upperDryingSectionGroup1FabricOverrunDriveSideAlarm := NOT P10_050_DI4.digitalInput_09,
    lowerDryingSectionGroup1FabricOverrunOperatorSideAlarm := NOT P10_050_DI4.digitalInput_16,
    lowerDryingSectionGroup1FabricOverrunDriveSideAlarm := NOT P10_050_DI4.digitalInput_15,
    dryingSectionGroup1PaperBreakAlarm := NOT P10_050_DI5.digitalInput_03,
    dryingSectionGroup2UpperMasterFaultAlarm := NOT P14_501_UG01_2GR_UpperMaster.statusWord.readyToSwitchOn,
    dryingSectionGroup2UpperSlave1FaultAlarm := NOT P13_501_UG02_2GR_UpperSlave.statusWord.readyToSwitchOn,
    dryingSectionGroup2LowerMasterFaultAlarm := NOT P13_501_UG03_2GR_LowerMaster.statusWord.readyToSwitchOn,
    dryingSectionGroup2LowerSlave1FaultAlarm := NOT P13_501_UG01_2GR_LowerSlave.statusWord.readyToSwitchOn,
    upperDryingSectionGroup2FabricOverrunOperatorSideAlarm := NOT P10_050_DI6.digitalInput_03,
    upperDryingSectionGroup2FabricOverrunDriveSideAlarm := NOT P10_050_DI6.digitalInput_02,
    lowerDryingSectionGroup2FabricOverrunOperatorSideAlarm := NOT P10_050_DI6.digitalInput_09,
    lowerDryingSectionGroup2FabricOverrunDriveSideAlarm := NOT P10_050_DI6.digitalInput_08,
    dryingSectionGroup3UpperMasterFaultAlarm := NOT P14_502_UG04_3GR_UpperMaster.statusWord.readyToSwitchOn,
    dryingSectionGroup3UpperSlave1FaultAlarm := NOT P14_502_UG02_3GR_UpperSlave.statusWord.readyToSwitchOn,
    dryingSectionGroup3LowerMasterFaultAlarm := NOT P14_502_UG03_3GR_LowerMaster.statusWord.readyToSwitchOn,
    dryingSectionGroup3LowerSlave1FaultAlarm := NOT P14_502_UG01_3GR_LowerSlave.statusWord.readyToSwitchOn,
    upperDryingSectionGroup3FabricOverrunOperatorSideAlarm := NOT P10_050_DI7.digitalInput_12,
    upperDryingSectionGroup3FabricOverrunDriveSideAlarm := NOT P10_050_DI7.digitalInput_11,
    lowerDryingSectionGroup3FabricOverrunOperatorSideAlarm := NOT P10_050_DI8.digitalInput_02,
    lowerDryingSectionGroup3FabricOverrunDriveSideAlarm := NOT P10_050_DI8.digitalInput_01,
    lubricationPump1FaultAlarm := NOT P10_050_DI8.digitalInput_09,
    lubricationPump2FaultAlarm := NOT P10_050_DI8.digitalInput_10,
    lubricationMinPressureFaultAlarm := NOT P10_050_DI8.digitalInput_13 AND P13_500_UG03_1GR_UpperMaster.commandWord.enableDrive,
    lubricationMaxPressureFaultAlarm := P10_050_DI8.digitalInput_12 AND P13_500_UG03_1GR_UpperMaster.commandWord.enableDrive,
    lubricationTankHighTemperatureAlarm := P10_050_AI2.Channel1 > 80,
    lubricationCircuitHighTemperatureAlarm := P10_050_AI2.Channel2 > 80,
    alarmIndication => paperMachineHmiStatus.alarmIndication); // FB_AlarmControl
paperMachineHmiAlarms := instFB_AlarmControl.alarmsDisplay;
END_METHOD

METHOD _CentrifugalPressureScreenControl
VAR_INPUT
END_VAR
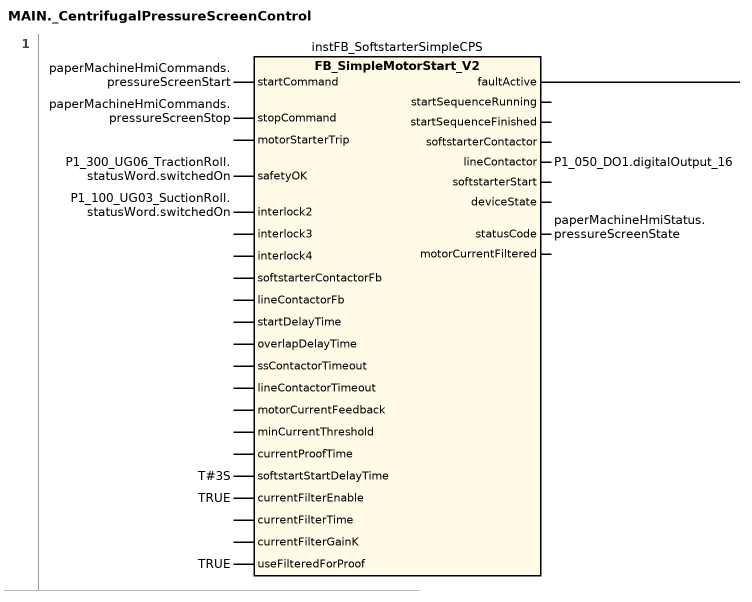
// NETWORK 1
instFB_SoftstarterSimpleCPS(
    startCommand := paperMachineHmiCommands.pressureScreenStart,
    stopCommand := paperMachineHmiCommands.pressureScreenStop,
    safetyOK := P1_300_UG06_TractionRoll.statusWord.switchedOn,
    interlock2 := P1_100_UG03_SuctionRoll.statusWord.switchedOn,
    softstartStartDelayTime := T#3S,
    currentFilterEnable := TRUE,
    useFilteredForProof := TRUE,
    lineContactor => P1_050_DO1.digitalOutput_16,
    statusCode => paperMachineHmiStatus.pressureScreenState); // FB_SimpleMotorStart_V2
END_METHOD

METHOD _CouchPitMixerControl
VAR_INPUT
END_VAR
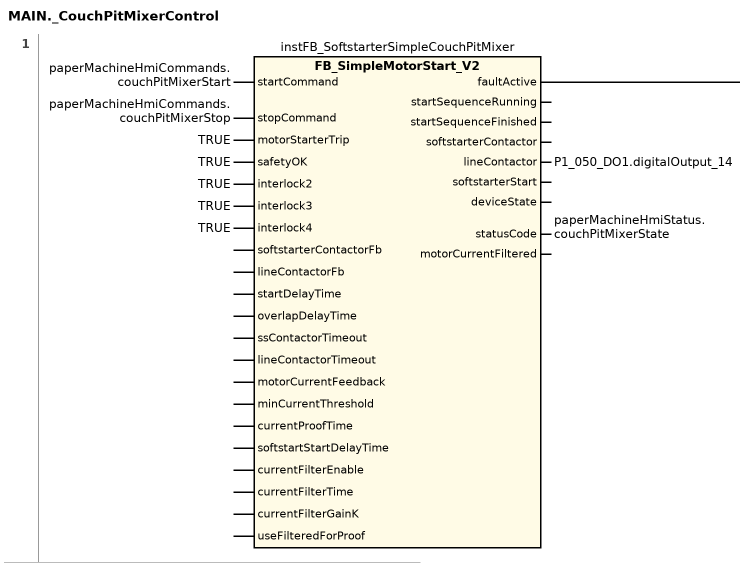
// NETWORK 1
instFB_SoftstarterSimpleCouchPitMixer(
    startCommand := paperMachineHmiCommands.couchPitMixerStart,
    stopCommand := paperMachineHmiCommands.couchPitMixerStop,
    motorStarterTrip := TRUE,
    safetyOK := TRUE,
    interlock2 := TRUE,
    interlock3 := TRUE,
    interlock4 := TRUE,
    lineContactor => P1_050_DO1.digitalOutput_14,
    statusCode => paperMachineHmiStatus.couchPitMixerState); // FB_SimpleMotorStart_V2
END_METHOD

METHOD _CouchPitPumpControl
VAR_INPUT
END_VAR
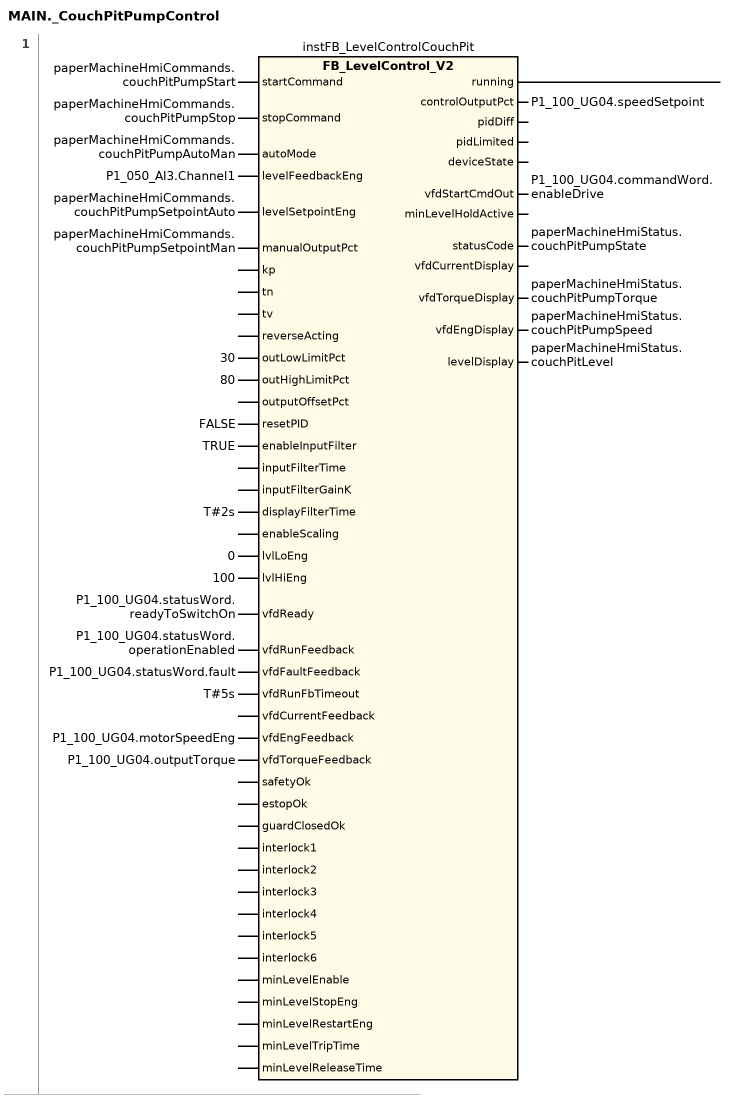
// NETWORK 1
instFB_LevelControlCouchPit(
    startCommand := paperMachineHmiCommands.couchPitPumpStart,
    stopCommand := paperMachineHmiCommands.couchPitPumpStop,
    autoMode := paperMachineHmiCommands.couchPitPumpAutoMan,
    levelFeedbackEng := P1_050_AI3.Channel1,
    levelSetpointEng := paperMachineHmiCommands.couchPitPumpSetpointAuto,
    manualOutputPct := paperMachineHmiCommands.couchPitPumpSetpointMan,
    outLowLimitPct := 30,
    outHighLimitPct := 80,
    resetPID := FALSE,
    enableInputFilter := TRUE,
    displayFilterTime := T#2s,
    lvlLoEng := 0,
    lvlHiEng := 100,
    vfdReady := P1_100_UG04.statusWord.readyToSwitchOn,
    vfdRunFeedback := P1_100_UG04.statusWord.operationEnabled,
    vfdFaultFeedback := P1_100_UG04.statusWord.fault,
    vfdRunFbTimeout := T#5s,
    vfdEngFeedback := P1_100_UG04.motorSpeedEng,
    vfdTorqueFeedback := P1_100_UG04.outputTorque,
    controlOutputPct => P1_100_UG04.speedSetpoint,
    vfdStartCmdOut => P1_100_UG04.commandWord.enableDrive,
    statusCode => paperMachineHmiStatus.couchPitPumpState,
    vfdTorqueDisplay => paperMachineHmiStatus.couchPitPumpTorque,
    vfdEngDisplay => paperMachineHmiStatus.couchPitPumpSpeed,
    levelDisplay => paperMachineHmiStatus.couchPitLevel); // FB_LevelControl_V2
END_METHOD

METHOD _FunctionBlockTest
VAR_INPUT
END_VAR
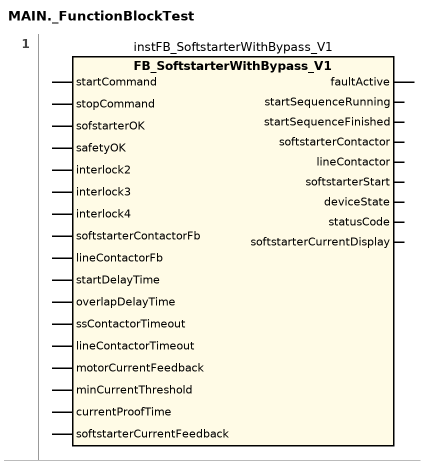
// NETWORK 1
instFB_SoftstarterWithBypass_V1(); // FB_SoftstarterWithBypass_V1
END_METHOD

METHOD _HeadBoxAuxiliaryControls
VAR_INPUT
END_VAR
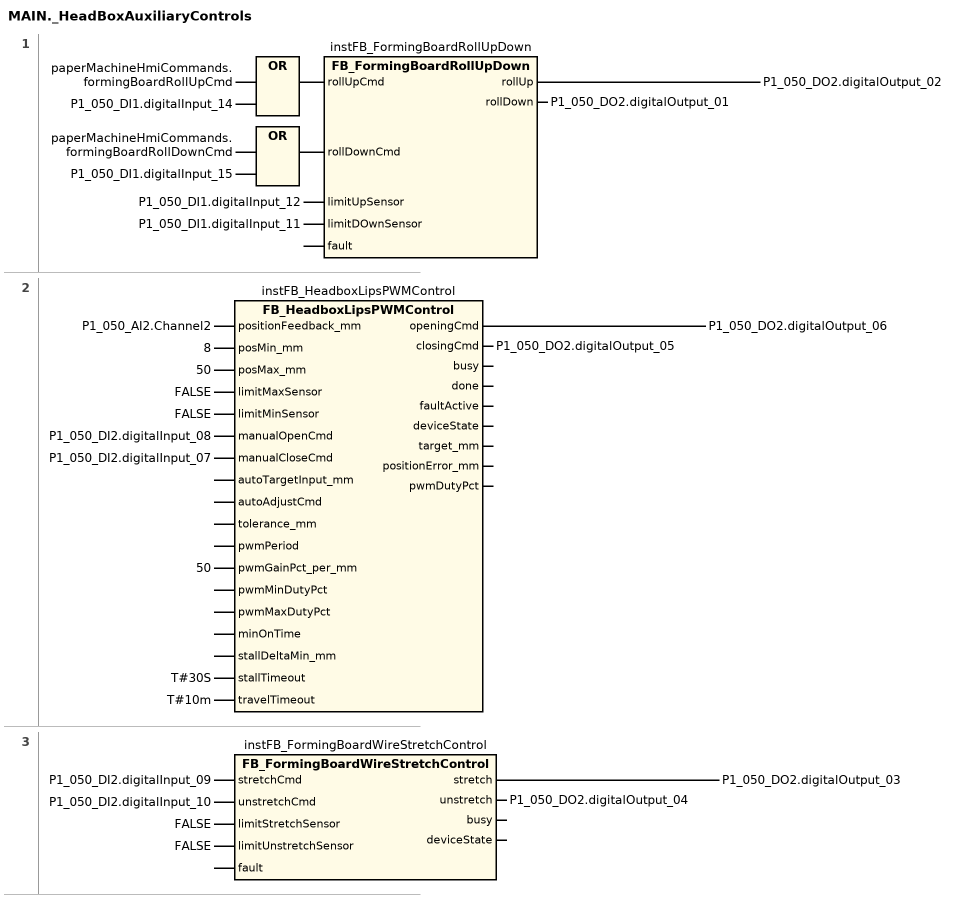
// NETWORK 1
instFB_FormingBoardRollUpDown(
    rollUpCmd := paperMachineHmiCommands.formingBoardRollUpCmd OR P1_050_DI1.digitalInput_14,
    rollDownCmd := paperMachineHmiCommands.formingBoardRollDownCmd OR P1_050_DI1.digitalInput_15,
    limitUpSensor := P1_050_DI1.digitalInput_12,
    limitDOwnSensor := P1_050_DI1.digitalInput_11,
    rollDown => P1_050_DO2.digitalOutput_01); // FB_FormingBoardRollUpDown
P1_050_DO2.digitalOutput_02 := instFB_FormingBoardRollUpDown.rollUp;

// NETWORK 2
instFB_HeadboxLipsPWMControl(
    positionFeedback_mm := P1_050_AI2.Channel2,
    posMin_mm := 8,
    posMax_mm := 50,
    limitMaxSensor := FALSE,
    limitMinSensor := FALSE,
    manualOpenCmd := P1_050_DI2.digitalInput_08,
    manualCloseCmd := P1_050_DI2.digitalInput_07,
    pwmGainPct_per_mm := 50,
    stallTimeout := T#30S,
    travelTimeout := T#10m,
    closingCmd => P1_050_DO2.digitalOutput_05); // FB_HeadboxLipsPWMControl
P1_050_DO2.digitalOutput_06 := instFB_HeadboxLipsPWMControl.openingCmd;

// NETWORK 3
instFB_FormingBoardWireStretchControl(
    stretchCmd := P1_050_DI2.digitalInput_09,
    unstretchCmd := P1_050_DI2.digitalInput_10,
    limitStretchSensor := FALSE,
    limitUnstretchSensor := FALSE,
    unstretch => P1_050_DO2.digitalOutput_04); // FB_FormingBoardWireStretchControl
P1_050_DO2.digitalOutput_03 := instFB_FormingBoardWireStretchControl.stretch;
END_METHOD

METHOD _MixPumpControl_1
VAR_INPUT
END_VAR
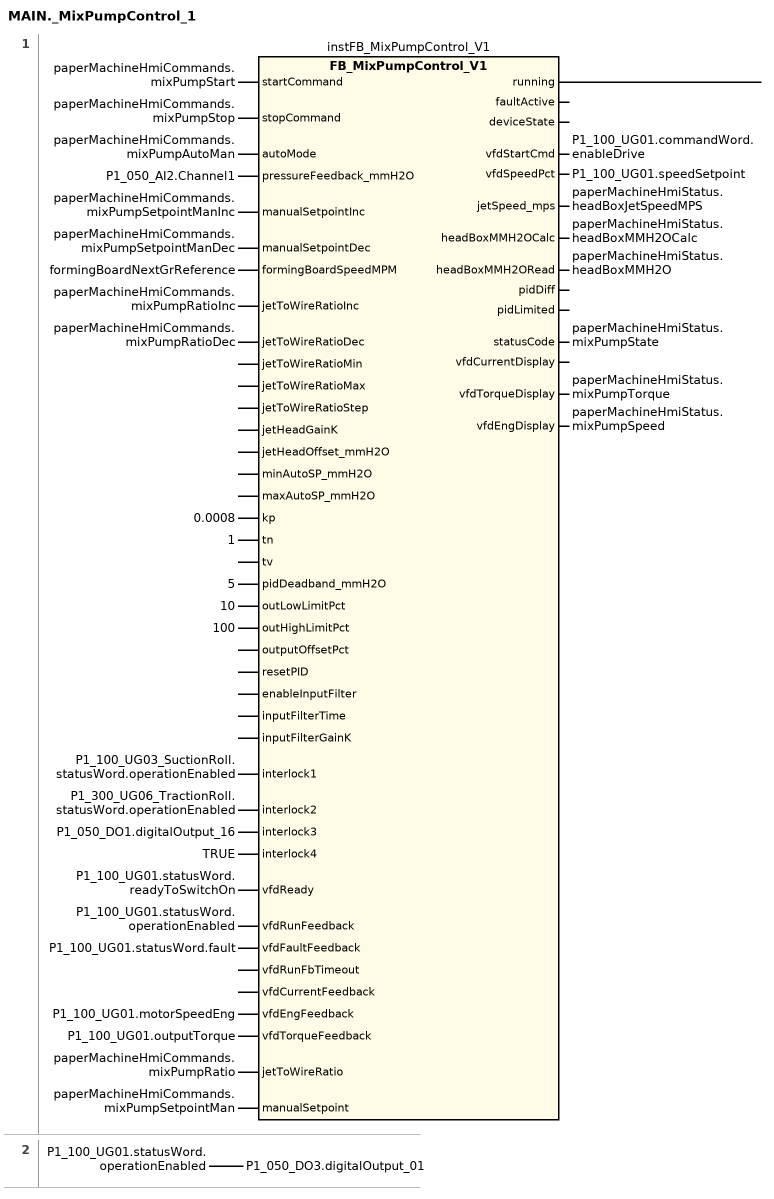
// NETWORK 1
instFB_MixPumpControl_V1(
    startCommand := paperMachineHmiCommands.mixPumpStart,
    stopCommand := paperMachineHmiCommands.mixPumpStop,
    autoMode := paperMachineHmiCommands.mixPumpAutoMan,
    pressureFeedback_mmH2O := P1_050_AI2.Channel1,
    manualSetpointInc := paperMachineHmiCommands.mixPumpSetpointManInc,
    manualSetpointDec := paperMachineHmiCommands.mixPumpSetpointManDec,
    formingBoardSpeedMPM := formingBoardNextGrReference,
    jetToWireRatioInc := paperMachineHmiCommands.mixPumpRatioInc,
    jetToWireRatioDec := paperMachineHmiCommands.mixPumpRatioDec,
    kp := 0.0008,
    tn := 1,
    pidDeadband_mmH2O := 5,
    outLowLimitPct := 10,
    outHighLimitPct := 100,
    interlock1 := P1_100_UG03_SuctionRoll.statusWord.operationEnabled,
    interlock2 := P1_300_UG06_TractionRoll.statusWord.operationEnabled,
    interlock3 := P1_050_DO1.digitalOutput_16,
    interlock4 := TRUE,
    vfdReady := P1_100_UG01.statusWord.readyToSwitchOn,
    vfdRunFeedback := P1_100_UG01.statusWord.operationEnabled,
    vfdFaultFeedback := P1_100_UG01.statusWord.fault,
    vfdEngFeedback := P1_100_UG01.motorSpeedEng,
    vfdTorqueFeedback := P1_100_UG01.outputTorque,
    jetToWireRatio := paperMachineHmiCommands.mixPumpRatio,
    manualSetpoint := paperMachineHmiCommands.mixPumpSetpointMan,
    vfdStartCmd => P1_100_UG01.commandWord.enableDrive,
    vfdSpeedPct => P1_100_UG01.speedSetpoint,
    jetSpeed_mps => paperMachineHmiStatus.headBoxJetSpeedMPS,
    headBoxMMH2OCalc => paperMachineHmiStatus.headBoxMMH2OCalc,
    headBoxMMH2ORead => paperMachineHmiStatus.headBoxMMH2O,
    statusCode => paperMachineHmiStatus.mixPumpState,
    vfdTorqueDisplay => paperMachineHmiStatus.mixPumpTorque,
    vfdEngDisplay => paperMachineHmiStatus.mixPumpSpeed); // FB_MixPumpControl_V1

// NETWORK 2
P1_050_DO3.digitalOutput_01 := P1_100_UG01.statusWord.operationEnabled;
END_METHOD

METHOD _StockPumpControl
VAR_INPUT
END_VAR

VAR
END_VAR
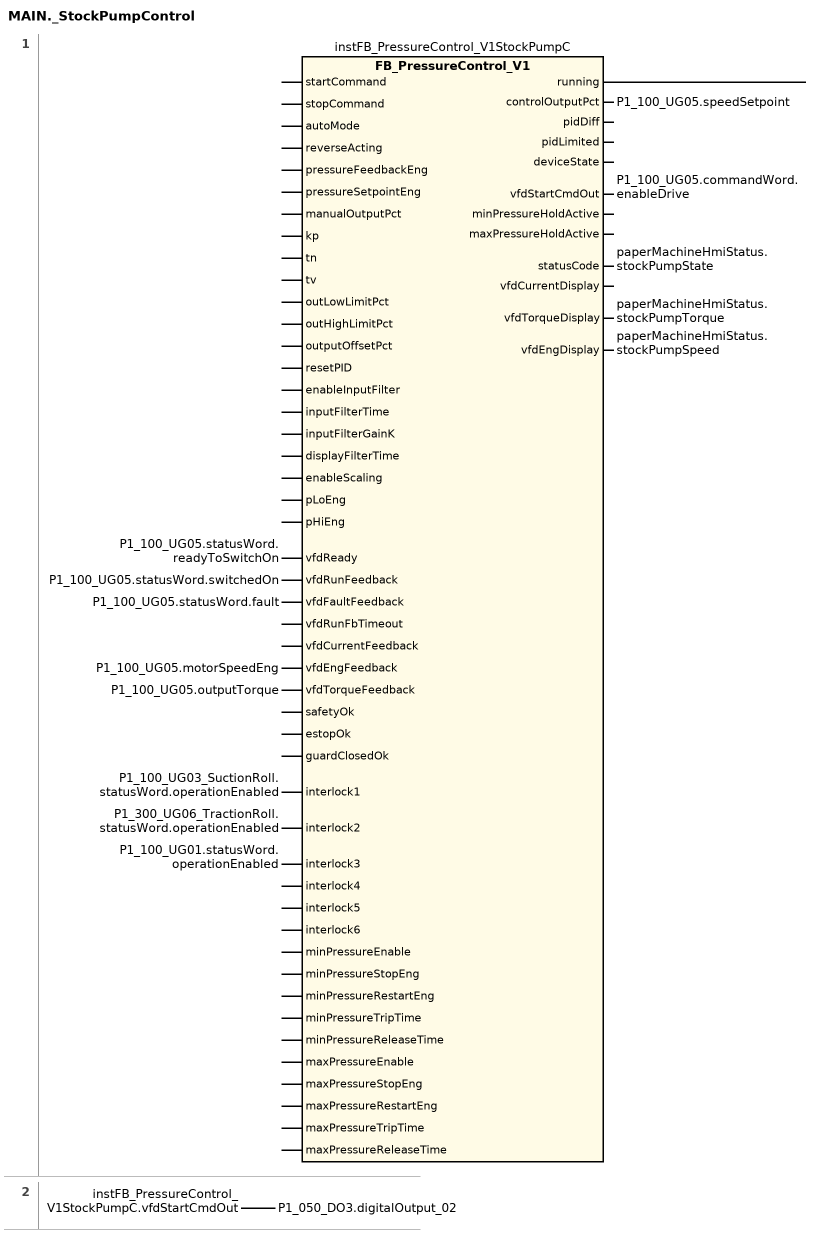
// NETWORK 1
instFB_PressureControl_V1StockPumpC(
    vfdReady := P1_100_UG05.statusWord.readyToSwitchOn,
    vfdRunFeedback := P1_100_UG05.statusWord.switchedOn,
    vfdFaultFeedback := P1_100_UG05.statusWord.fault,
    vfdEngFeedback := P1_100_UG05.motorSpeedEng,
    vfdTorqueFeedback := P1_100_UG05.outputTorque,
    interlock1 := P1_100_UG03_SuctionRoll.statusWord.operationEnabled,
    interlock2 := P1_300_UG06_TractionRoll.statusWord.operationEnabled,
    interlock3 := P1_100_UG01.statusWord.operationEnabled,
    controlOutputPct => P1_100_UG05.speedSetpoint,
    vfdStartCmdOut => P1_100_UG05.commandWord.enableDrive,
    statusCode => paperMachineHmiStatus.stockPumpState,
    vfdTorqueDisplay => paperMachineHmiStatus.stockPumpTorque,
    vfdEngDisplay => paperMachineHmiStatus.stockPumpSpeed); // FB_PressureControl_V1

// NETWORK 2
P1_050_DO3.digitalOutput_02 := instFB_PressureControl_V1StockPumpC.vfdStartCmdOut;
END_METHOD

METHOD _StockPumpControl_1
VAR_INPUT
END_VAR

VAR
END_VAR
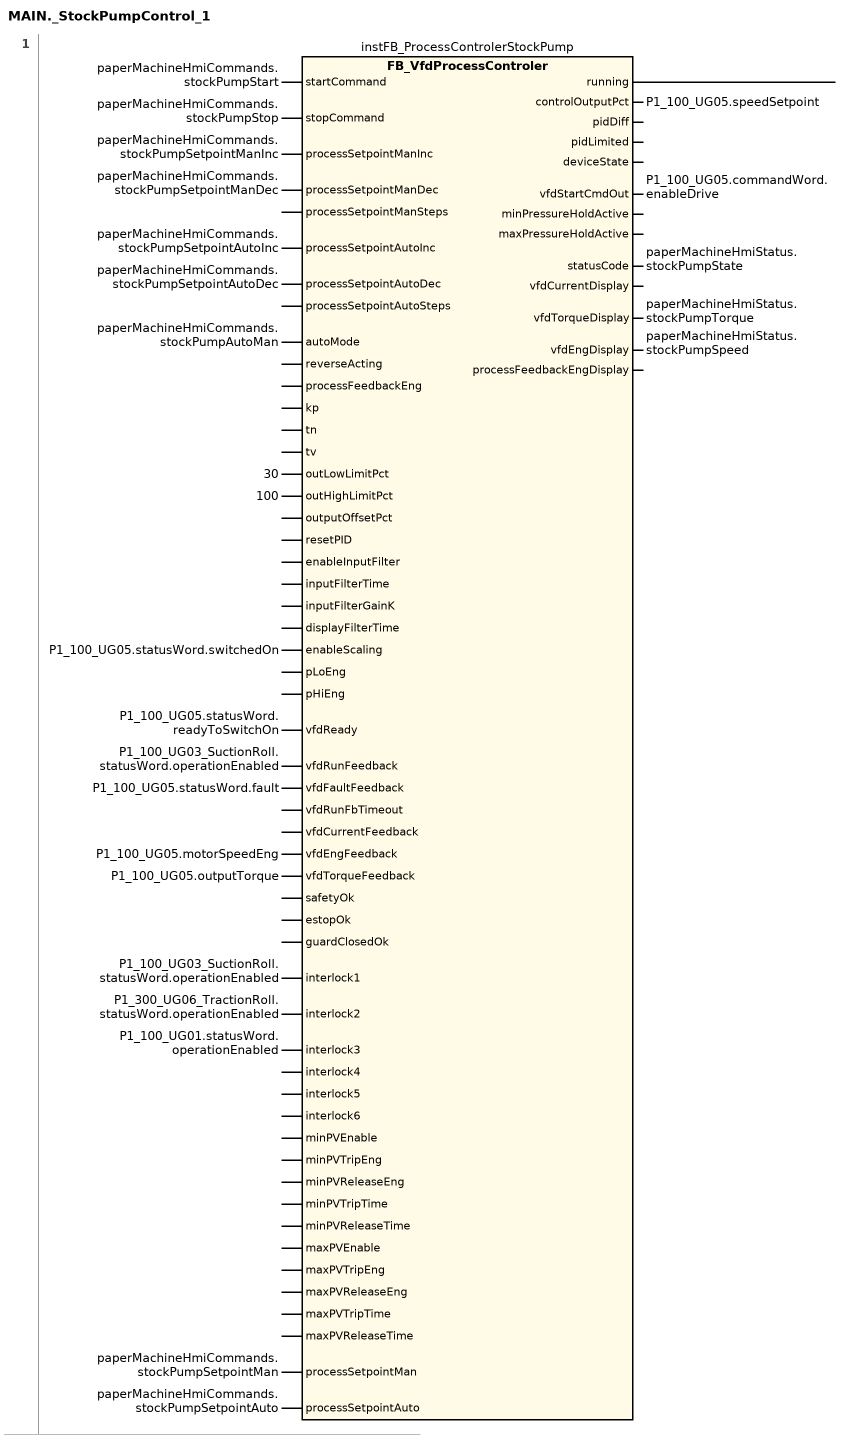
// NETWORK 1
instFB_ProcessControlerStockPump(
    startCommand := paperMachineHmiCommands.stockPumpStart,
    stopCommand := paperMachineHmiCommands.stockPumpStop,
    processSetpointManInc := paperMachineHmiCommands.stockPumpSetpointManInc,
    processSetpointManDec := paperMachineHmiCommands.stockPumpSetpointManDec,
    processSetpointAutoInc := paperMachineHmiCommands.stockPumpSetpointAutoInc,
    processSetpointAutoDec := paperMachineHmiCommands.stockPumpSetpointAutoDec,
    autoMode := paperMachineHmiCommands.stockPumpAutoMan,
    outLowLimitPct := 30,
    outHighLimitPct := 100,
    enableScaling := P1_100_UG05.statusWord.switchedOn,
    vfdReady := P1_100_UG05.statusWord.readyToSwitchOn,
    vfdRunFeedback := P1_100_UG03_SuctionRoll.statusWord.operationEnabled,
    vfdFaultFeedback := P1_100_UG05.statusWord.fault,
    vfdEngFeedback := P1_100_UG05.motorSpeedEng,
    vfdTorqueFeedback := P1_100_UG05.outputTorque,
    interlock1 := P1_100_UG03_SuctionRoll.statusWord.operationEnabled,
    interlock2 := P1_300_UG06_TractionRoll.statusWord.operationEnabled,
    interlock3 := P1_100_UG01.statusWord.operationEnabled,
    processSetpointMan := paperMachineHmiCommands.stockPumpSetpointMan,
    processSetpointAuto := paperMachineHmiCommands.stockPumpSetpointAuto,
    controlOutputPct => P1_100_UG05.speedSetpoint,
    vfdStartCmdOut => P1_100_UG05.commandWord.enableDrive,
    statusCode => paperMachineHmiStatus.stockPumpState,
    vfdTorqueDisplay => paperMachineHmiStatus.stockPumpTorque,
    vfdEngDisplay => paperMachineHmiStatus.stockPumpSpeed); // FB_VfdProcessControler

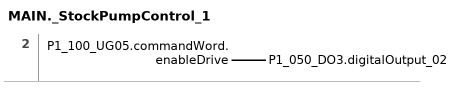
// NETWORK 2
P1_050_DO3.digitalOutput_02 := P1_100_UG05.commandWord.enableDrive;
END_METHOD

METHOD _VaccumPumps
VAR_INPUT
END_VAR
(*

    // ─────────────── LOW VACUUM EXHAUST FAN ───────────────
    lowVacuumExhaustFanStart : BOOL;  // Start low vacuum exhaust fan (Ligar exaustor do baixo vácuo)
    lowVacuumExhaustFanStop  : BOOL;  // Stop low vacuum exhaust fan (Parar exaustor do baixo vácuo)
	
	paperMachineHmiCommands.suctionRollVacuumPumpStart
	paperMachineHmiCommands.suctionRollVacuumPumpStop
	paperMachineHmiCommands.wireVacuumPumpStart
	paperMachineHmiCommands.wireVacuumPumpStop


*)
VAR_INST // added by the converter: edge detectors and wires of the graphical bodies
    _w1 : BOOL;
END_VAR
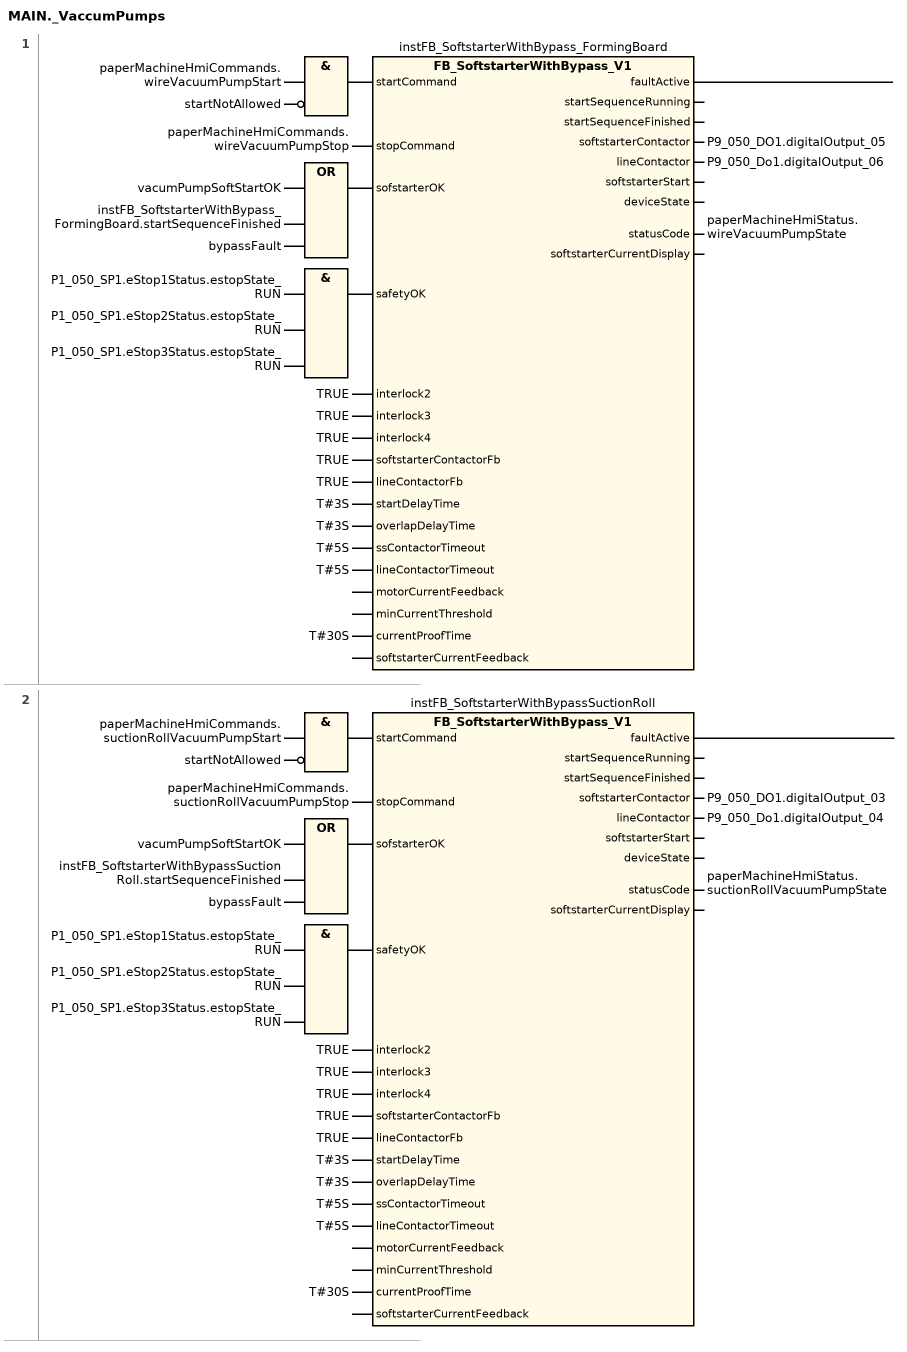
// NETWORK 1
instFB_SoftstarterWithBypass_FormingBoard(
    startCommand := paperMachineHmiCommands.wireVacuumPumpStart AND NOT startNotAllowed,
    stopCommand := paperMachineHmiCommands.wireVacuumPumpStop,
    sofstarterOK := vacumPumpSoftStartOK OR instFB_SoftstarterWithBypass_FormingBoard.startSequenceFinished OR bypassFault,
    safetyOK := P1_050_SP1.eStop1Status.estopState_RUN AND P1_050_SP1.eStop2Status.estopState_RUN AND P1_050_SP1.eStop3Status.estopState_RUN,
    interlock2 := TRUE,
    interlock3 := TRUE,
    interlock4 := TRUE,
    softstarterContactorFb := TRUE,
    lineContactorFb := TRUE,
    startDelayTime := T#3S,
    overlapDelayTime := T#3S,
    ssContactorTimeout := T#5S,
    lineContactorTimeout := T#5S,
    currentProofTime := T#30S,
    softstarterContactor => P9_050_DO1.digitalOutput_05,
    lineContactor => P9_050_Do1.digitalOutput_06,
    statusCode => paperMachineHmiStatus.wireVacuumPumpState); // FB_SoftstarterWithBypass_V1

// NETWORK 2
instFB_SoftstarterWithBypassSuctionRoll(
    startCommand := paperMachineHmiCommands.suctionRollVacuumPumpStart AND NOT startNotAllowed,
    stopCommand := paperMachineHmiCommands.suctionRollVacuumPumpStop,
    sofstarterOK := vacumPumpSoftStartOK OR instFB_SoftstarterWithBypassSuctionRoll.startSequenceFinished OR bypassFault,
    safetyOK := P1_050_SP1.eStop1Status.estopState_RUN AND P1_050_SP1.eStop2Status.estopState_RUN AND P1_050_SP1.eStop3Status.estopState_RUN,
    interlock2 := TRUE,
    interlock3 := TRUE,
    interlock4 := TRUE,
    softstarterContactorFb := TRUE,
    lineContactorFb := TRUE,
    startDelayTime := T#3S,
    overlapDelayTime := T#3S,
    ssContactorTimeout := T#5S,
    lineContactorTimeout := T#5S,
    currentProofTime := T#30S,
    softstarterContactor => P9_050_DO1.digitalOutput_03,
    lineContactor => P9_050_Do1.digitalOutput_04,
    statusCode => paperMachineHmiStatus.suctionRollVacuumPumpState); // FB_SoftstarterWithBypass_V1

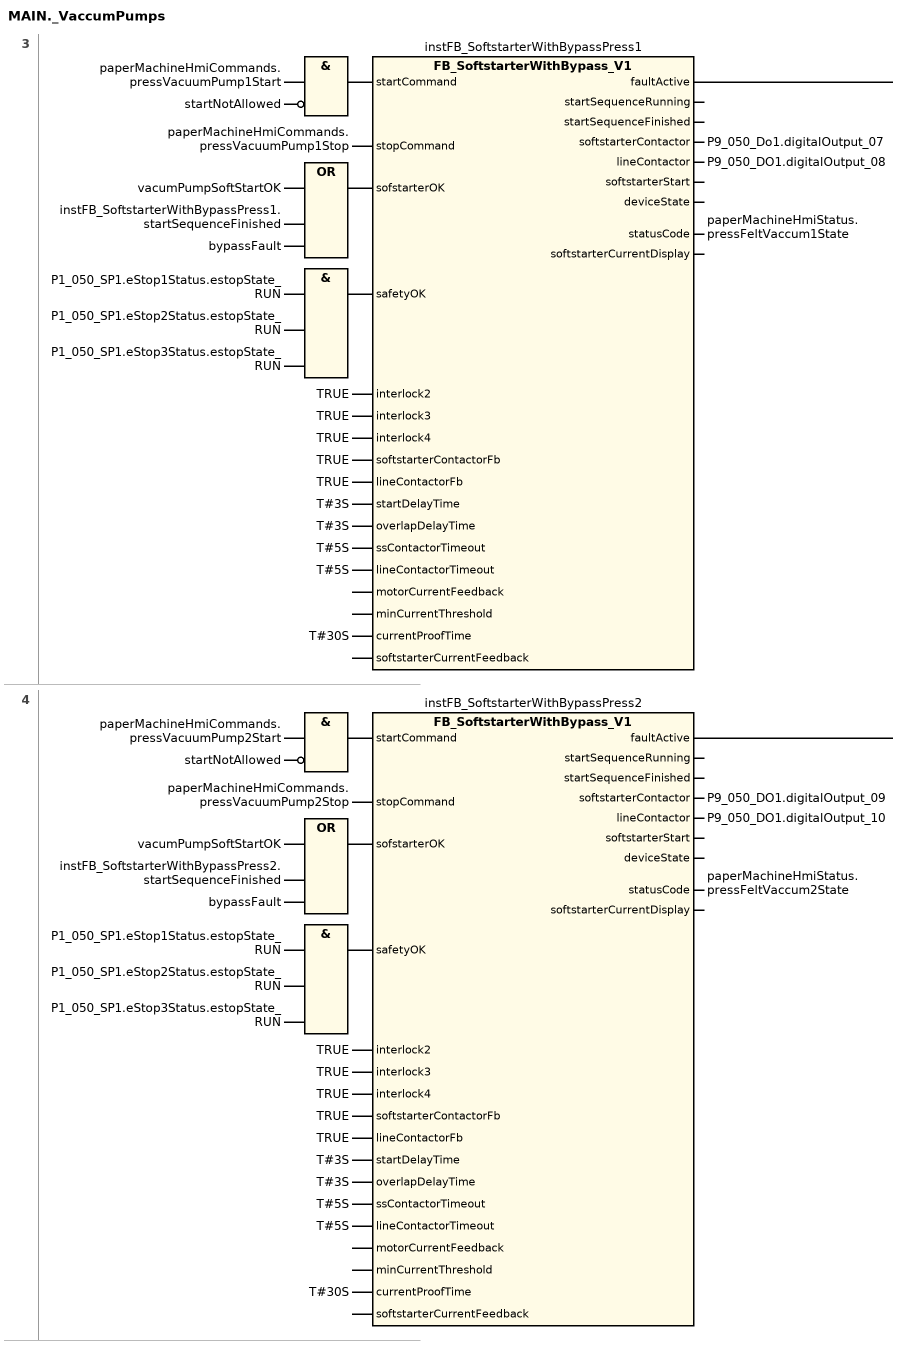
// NETWORK 3
instFB_SoftstarterWithBypassPress1(
    startCommand := paperMachineHmiCommands.pressVacuumPump1Start AND NOT startNotAllowed,
    stopCommand := paperMachineHmiCommands.pressVacuumPump1Stop,
    sofstarterOK := vacumPumpSoftStartOK OR instFB_SoftstarterWithBypassPress1.startSequenceFinished OR bypassFault,
    safetyOK := P1_050_SP1.eStop1Status.estopState_RUN AND P1_050_SP1.eStop2Status.estopState_RUN AND P1_050_SP1.eStop3Status.estopState_RUN,
    interlock2 := TRUE,
    interlock3 := TRUE,
    interlock4 := TRUE,
    softstarterContactorFb := TRUE,
    lineContactorFb := TRUE,
    startDelayTime := T#3S,
    overlapDelayTime := T#3S,
    ssContactorTimeout := T#5S,
    lineContactorTimeout := T#5S,
    currentProofTime := T#30S,
    softstarterContactor => P9_050_Do1.digitalOutput_07,
    lineContactor => P9_050_DO1.digitalOutput_08,
    statusCode => paperMachineHmiStatus.pressFeltVaccum1State); // FB_SoftstarterWithBypass_V1

// NETWORK 4
instFB_SoftstarterWithBypassPress2(
    startCommand := paperMachineHmiCommands.pressVacuumPump2Start AND NOT startNotAllowed,
    stopCommand := paperMachineHmiCommands.pressVacuumPump2Stop,
    sofstarterOK := vacumPumpSoftStartOK OR instFB_SoftstarterWithBypassPress2.startSequenceFinished OR bypassFault,
    safetyOK := P1_050_SP1.eStop1Status.estopState_RUN AND P1_050_SP1.eStop2Status.estopState_RUN AND P1_050_SP1.eStop3Status.estopState_RUN,
    interlock2 := TRUE,
    interlock3 := TRUE,
    interlock4 := TRUE,
    softstarterContactorFb := TRUE,
    lineContactorFb := TRUE,
    startDelayTime := T#3S,
    overlapDelayTime := T#3S,
    ssContactorTimeout := T#5S,
    lineContactorTimeout := T#5S,
    currentProofTime := T#30S,
    softstarterContactor => P9_050_DO1.digitalOutput_09,
    lineContactor => P9_050_DO1.digitalOutput_10,
    statusCode => paperMachineHmiStatus.pressFeltVaccum2State); // FB_SoftstarterWithBypass_V1

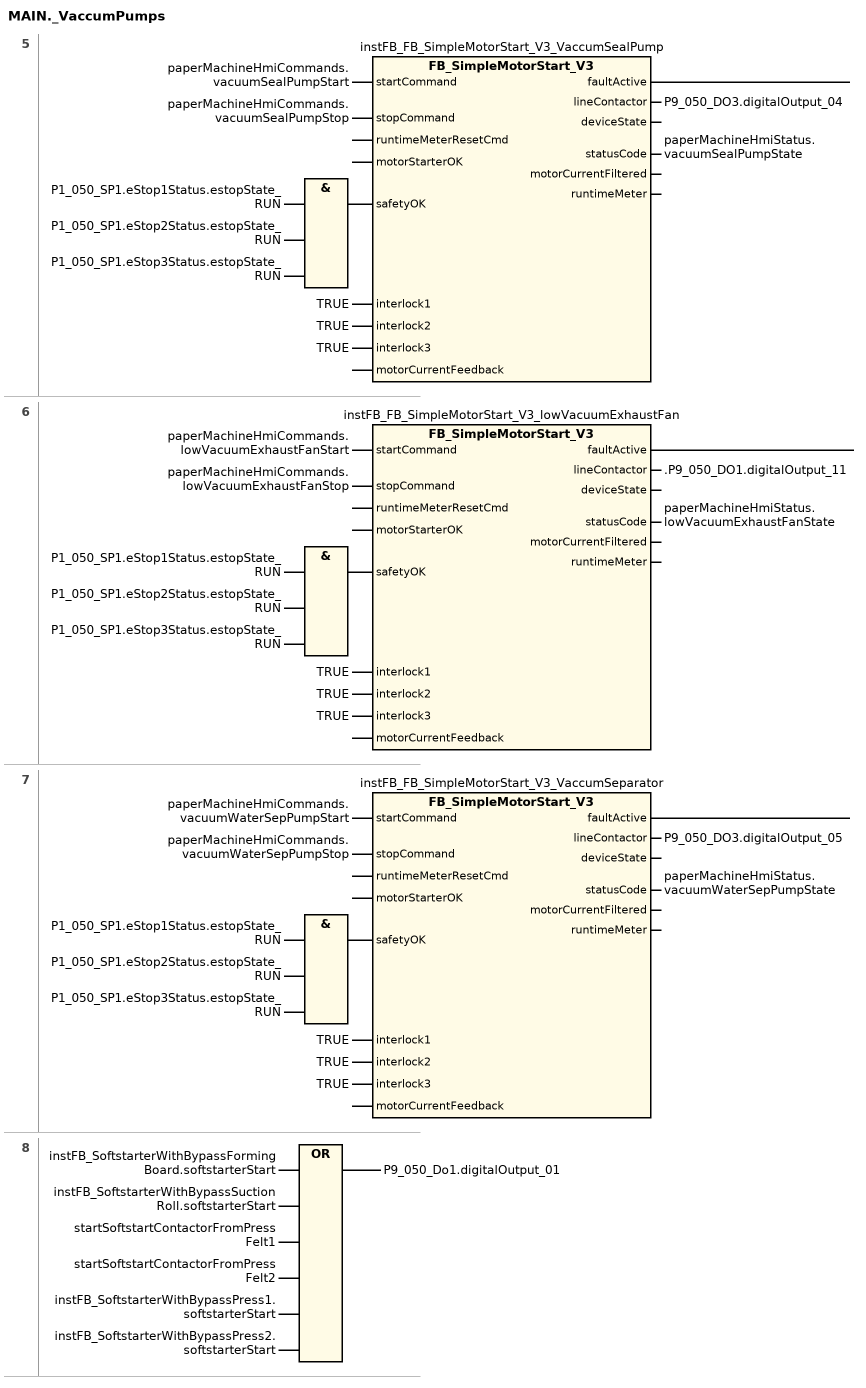
// NETWORK 5
instFB_FB_SimpleMotorStart_V3_VaccumSealPump(
    startCommand := paperMachineHmiCommands.vacuumSealPumpStart,
    stopCommand := paperMachineHmiCommands.vacuumSealPumpStop,
    safetyOK := P1_050_SP1.eStop1Status.estopState_RUN AND P1_050_SP1.eStop2Status.estopState_RUN AND P1_050_SP1.eStop3Status.estopState_RUN,
    interlock1 := TRUE,
    interlock2 := TRUE,
    interlock3 := TRUE,
    lineContactor => P9_050_DO3.digitalOutput_04,
    statusCode => paperMachineHmiStatus.vacuumSealPumpState); // FB_SimpleMotorStart_V3

// NETWORK 6
instFB_FB_SimpleMotorStart_V3_lowVacuumExhaustFan(
    startCommand := paperMachineHmiCommands.lowVacuumExhaustFanStart,
    stopCommand := paperMachineHmiCommands.lowVacuumExhaustFanStop,
    safetyOK := P1_050_SP1.eStop1Status.estopState_RUN AND P1_050_SP1.eStop2Status.estopState_RUN AND P1_050_SP1.eStop3Status.estopState_RUN,
    interlock1 := TRUE,
    interlock2 := TRUE,
    interlock3 := TRUE,
    lineContactor => .P9_050_DO1.digitalOutput_11,
    statusCode => paperMachineHmiStatus.lowVacuumExhaustFanState); // FB_SimpleMotorStart_V3

// NETWORK 7
instFB_FB_SimpleMotorStart_V3_VaccumSeparator(
    startCommand := paperMachineHmiCommands.vacuumWaterSepPumpStart,
    stopCommand := paperMachineHmiCommands.vacuumWaterSepPumpStop,
    safetyOK := P1_050_SP1.eStop1Status.estopState_RUN AND P1_050_SP1.eStop2Status.estopState_RUN AND P1_050_SP1.eStop3Status.estopState_RUN,
    interlock1 := TRUE,
    interlock2 := TRUE,
    interlock3 := TRUE,
    lineContactor => P9_050_DO3.digitalOutput_05,
    statusCode => paperMachineHmiStatus.vacuumWaterSepPumpState); // FB_SimpleMotorStart_V3

// NETWORK 8
P9_050_Do1.digitalOutput_01 := instFB_SoftstarterWithBypassFormingBoard.softstarterStart OR instFB_SoftstarterWithBypassSuctionRoll.softstarterStart OR startSoftstartContactorFromPressFelt1 OR startSoftstartContactorFromPressFelt2 OR instFB_SoftstarterWithBypassPress1.softstarterStart OR instFB_SoftstarterWithBypassPress2.softstarterStart;

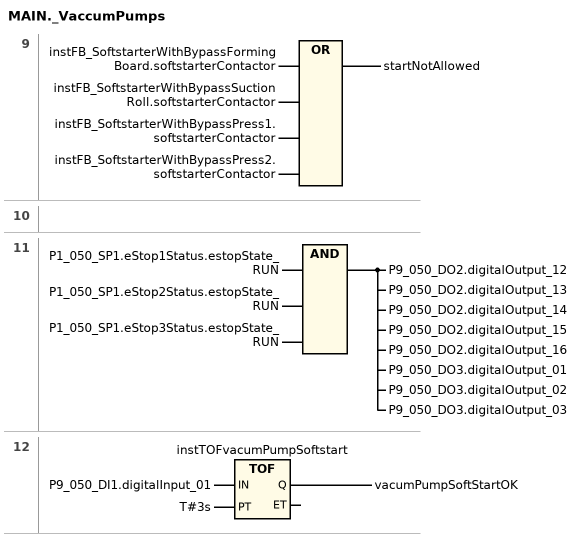
// NETWORK 9
startNotAllowed := instFB_SoftstarterWithBypassFormingBoard.softstarterContactor OR instFB_SoftstarterWithBypassSuctionRoll.softstarterContactor OR instFB_SoftstarterWithBypassPress1.softstarterContactor OR instFB_SoftstarterWithBypassPress2.softstarterContactor;

// NETWORK 10

// NETWORK 11
_w1 := P1_050_SP1.eStop1Status.estopState_RUN AND P1_050_SP1.eStop2Status.estopState_RUN AND P1_050_SP1.eStop3Status.estopState_RUN;
P9_050_DO2.digitalOutput_12 := _w1;
P9_050_DO2.digitalOutput_13 := _w1;
P9_050_DO2.digitalOutput_14 := _w1;
P9_050_DO2.digitalOutput_15 := _w1;
P9_050_DO2.digitalOutput_16 := _w1;
P9_050_DO3.digitalOutput_01 := _w1;
P9_050_DO3.digitalOutput_02 := _w1;
P9_050_DO3.digitalOutput_03 := _w1;

// NETWORK 12
instTOFvacumPumpSoftstart(IN := P9_050_DI1.digitalInput_01, PT := T#3s); // TOF
vacumPumpSoftStartOK := instTOFvacumPumpSoftstart.Q;
END_METHOD

METHOD _WirePitControl
VAR_INPUT
END_VAR
//P1_050_AI4.Channel1
(*

paperMachineHmiCommands.whiteWaterSiloSetpointMan
paperMachineHmiCommands.whiteWaterSiloSetpointAuto
paperMachineHmiCommands.wirePitSetpointMan
paperMachineHmiCommands.wirePitSetpointAuto
*)
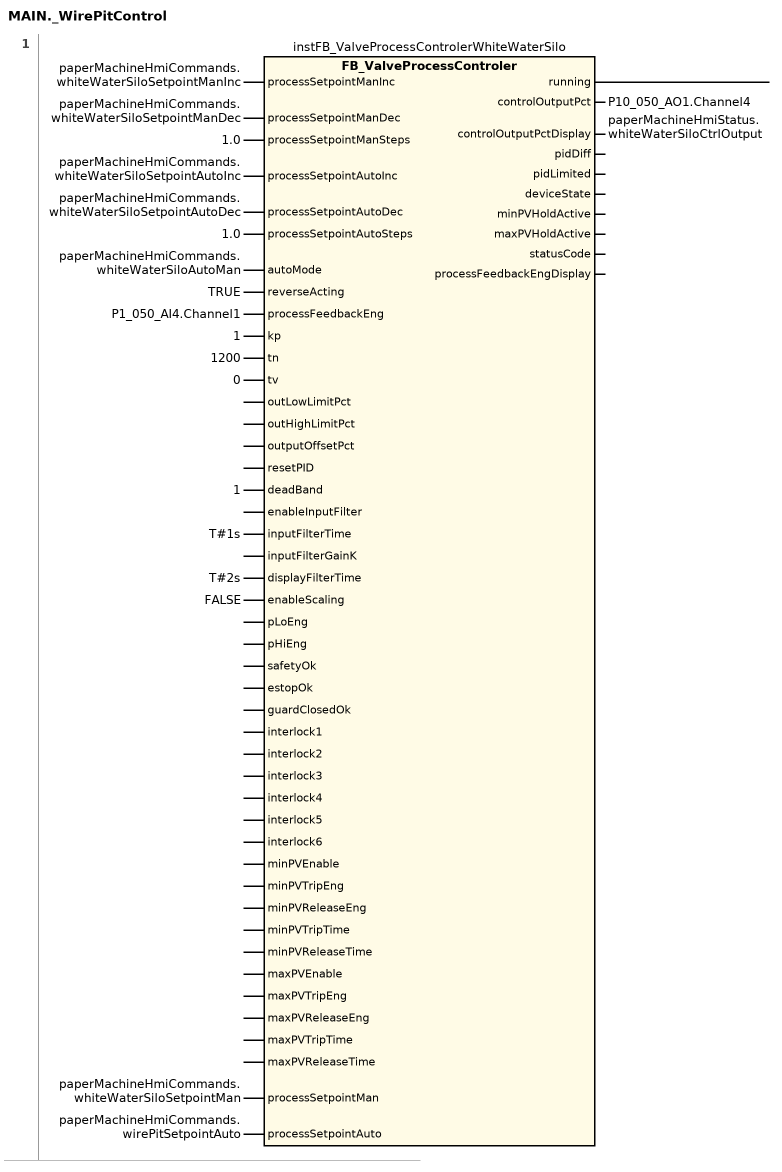
// NETWORK 1
instFB_ValveProcessControlerWhiteWaterSilo(
    processSetpointManInc := paperMachineHmiCommands.whiteWaterSiloSetpointManInc,
    processSetpointManDec := paperMachineHmiCommands.whiteWaterSiloSetpointManDec,
    processSetpointManSteps := 1.0,
    processSetpointAutoInc := paperMachineHmiCommands.whiteWaterSiloSetpointAutoInc,
    processSetpointAutoDec := paperMachineHmiCommands.whiteWaterSiloSetpointAutoDec,
    processSetpointAutoSteps := 1.0,
    autoMode := paperMachineHmiCommands.whiteWaterSiloAutoMan,
    reverseActing := TRUE,
    processFeedbackEng := P1_050_AI4.Channel1,
    kp := 1,
    tn := 1200,
    tv := 0,
    deadBand := 1,
    inputFilterTime := T#1s,
    displayFilterTime := T#2s,
    enableScaling := FALSE,
    processSetpointMan := paperMachineHmiCommands.whiteWaterSiloSetpointMan,
    processSetpointAuto := paperMachineHmiCommands.wirePitSetpointAuto,
    controlOutputPct => P10_050_AO1.Channel4,
    controlOutputPctDisplay => paperMachineHmiStatus.whiteWaterSiloCtrlOutput); // FB_ValveProcessControler

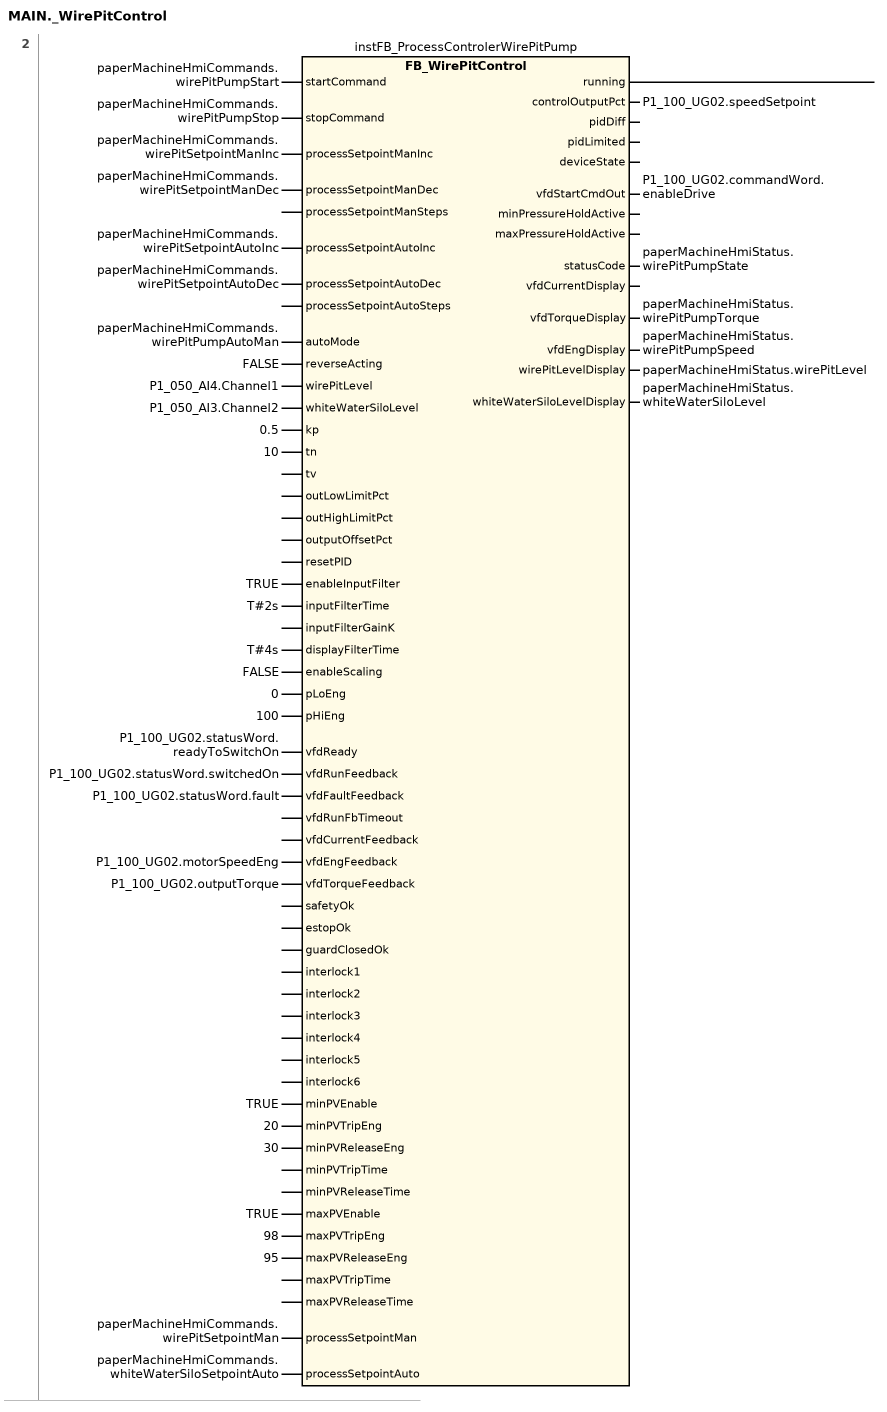
// NETWORK 2
instFB_ProcessControlerWirePitPump(
    startCommand := paperMachineHmiCommands.wirePitPumpStart,
    stopCommand := paperMachineHmiCommands.wirePitPumpStop,
    processSetpointManInc := paperMachineHmiCommands.wirePitSetpointManInc,
    processSetpointManDec := paperMachineHmiCommands.wirePitSetpointManDec,
    processSetpointAutoInc := paperMachineHmiCommands.wirePitSetpointAutoInc,
    processSetpointAutoDec := paperMachineHmiCommands.wirePitSetpointAutoDec,
    autoMode := paperMachineHmiCommands.wirePitPumpAutoMan,
    reverseActing := FALSE,
    wirePitLevel := P1_050_AI4.Channel1,
    whiteWaterSiloLevel := P1_050_AI3.Channel2,
    kp := 0.5,
    tn := 10,
    enableInputFilter := TRUE,
    inputFilterTime := T#2s,
    displayFilterTime := T#4s,
    enableScaling := FALSE,
    pLoEng := 0,
    pHiEng := 100,
    vfdReady := P1_100_UG02.statusWord.readyToSwitchOn,
    vfdRunFeedback := P1_100_UG02.statusWord.switchedOn,
    vfdFaultFeedback := P1_100_UG02.statusWord.fault,
    vfdEngFeedback := P1_100_UG02.motorSpeedEng,
    vfdTorqueFeedback := P1_100_UG02.outputTorque,
    minPVEnable := TRUE,
    minPVTripEng := 20,
    minPVReleaseEng := 30,
    maxPVEnable := TRUE,
    maxPVTripEng := 98,
    maxPVReleaseEng := 95,
    processSetpointMan := paperMachineHmiCommands.wirePitSetpointMan,
    processSetpointAuto := paperMachineHmiCommands.whiteWaterSiloSetpointAuto,
    controlOutputPct => P1_100_UG02.speedSetpoint,
    vfdStartCmdOut => P1_100_UG02.commandWord.enableDrive,
    statusCode => paperMachineHmiStatus.wirePitPumpState,
    vfdTorqueDisplay => paperMachineHmiStatus.wirePitPumpTorque,
    vfdEngDisplay => paperMachineHmiStatus.wirePitPumpSpeed,
    wirePitLevelDisplay => paperMachineHmiStatus.wirePitLevel,
    whiteWaterSiloLevelDisplay => paperMachineHmiStatus.whiteWaterSiloLevel); // FB_WirePitControl
END_METHOD

METHOD machineReset
VAR_INPUT
END_VAR

VAR
	instTP_Reset: TP;
END_VAR
//────────────────────────────────────────────
// UG01 to UG06 (General Utilities / Aux Drives)
//────────────────────────────────────────────
P1_100_UG01.commandWord.faultResetCmd := paperMachineHmiCommands.machineReset;
P1_100_UG02.commandWord.faultResetCmd := paperMachineHmiCommands.machineReset;
P1_100_UG03_SuctionRoll.commandWord.faultResetCmd := paperMachineHmiCommands.machineReset;
P1_100_UG04.commandWord.faultResetCmd := paperMachineHmiCommands.machineReset;
P1_100_UG05.commandWord.faultResetCmd := paperMachineHmiCommands.machineReset;
P1_300_UG06_TractionRoll.commandWord.faultResetCmd := paperMachineHmiCommands.machineReset;

//────────────────────────────────────────────
// Safety PLC Reset
//────────────────────────────────────────────
P1_050_SP1.safetyReset := paperMachineHmiCommands.machineReset;
P1_050_SP1.errorAcknowledgement := paperMachineHmiCommands.machineReset;

//────────────────────────────────────────────
// Press Section Drives
//────────────────────────────────────────────
P11_400_UG01_SecondPress.commandWord.faultResetCmd := paperMachineHmiCommands.machineReset;
P12_400_UG01_FirstPress.commandWord.faultResetCmd := paperMachineHmiCommands.machineReset;

//────────────────────────────────────────────
// Drying Section — Group 1
//────────────────────────────────────────────
P13_500_UG01_1GR_UpperSlave.commandWord.faultResetCmd := paperMachineHmiCommands.machineReset;
P13_500_UG02_1GR_LowerMaster.commandWord.faultResetCmd := paperMachineHmiCommands.machineReset;
P13_500_UG03_1GR_UpperMaster.commandWord.faultResetCmd := paperMachineHmiCommands.machineReset;

//────────────────────────────────────────────
// Drying Section — Group 2
//────────────────────────────────────────────
P13_501_UG01_2GR_LowerSlave.commandWord.faultResetCmd := paperMachineHmiCommands.machineReset;
P13_501_UG02_2GR_UpperSlave.commandWord.faultResetCmd := paperMachineHmiCommands.machineReset;
P13_501_UG03_2GR_LowerMaster.commandWord.faultResetCmd := paperMachineHmiCommands.machineReset;
P14_501_UG01_2GR_UpperMaster.commandWord.faultResetCmd := paperMachineHmiCommands.machineReset;

//────────────────────────────────────────────
// Drying Section — Group 3
//────────────────────────────────────────────
P14_502_UG01_3GR_LowerSlave.commandWord.faultResetCmd := paperMachineHmiCommands.machineReset;
P14_502_UG02_3GR_UpperSlave.commandWord.faultResetCmd := paperMachineHmiCommands.machineReset;
P14_502_UG03_3GR_LowerMaster.commandWord.faultResetCmd := paperMachineHmiCommands.machineReset;
P14_502_UG04_3GR_UpperMaster.commandWord.faultResetCmd := paperMachineHmiCommands.machineReset;

//────────────────────────────────────────────
// Rewinder
//────────────────────────────────────────────
P15_600_UG01_Rewinder.commandWord.faultResetCmd := paperMachineHmiCommands.machineReset;
END_METHOD

END_PROGRAM

// ---- Function Blocks/PaperMachine/DriveControl/FB_DryingSectionLubrificationControl_V1.TcPOU
FUNCTION_BLOCK FB_DryingSectionLubrificationControl_V1
VAR_INPUT
    //==============================================================
    // COMMANDS / INTERLOCKS
    //==============================================================
    startCmd               : BOOL;    // EN: Manual start command / PT: Comando de partida manual
    stopCmd                : BOOL;    // EN: Manual stop command / PT: Comando de parada manual
    machineRunningFeedback : BOOL;    // EN: Machine running feedback / PT: Sinal de máquina em operação
    pumpSelector           : BOOL;    // EN: Pump selector (FALSE = Pump1 / TRUE = Pump2) / PT: Seletor de bomba (FALSE = B1 / TRUE = B2)

	pump1Fault				: BOOL;
	pump2Fault				: BOOL;	

	minPressureFeedback		: BOOL;
	maxPressureFeedback		: BOOL;		
	
    //==============================================================
    // TEMPERATURE MEASUREMENT
    //==============================================================
    tankTemperature        : REAL;    // EN: Lubrication oil tank temperature [°C] / PT: Temperatura do tanque de óleo [°C]
    circuitTemperature     : REAL;    // EN: Lubrication circuit temperature [°C] / PT: Temperatura do circuito de lubrificação [°C]

	
    tankMaxTemperature        : REAL := 60.0;    // EN: Lubrication oil tank temperature [°C] / PT: Temperatura do tanque de óleo [°C]
    circuitMaxTemperature     : REAL := 65.0;    // EN: Lubrication circuit temperature [°C] / PT: Temperatura do circuito de lubrificação [°C]
	
	
    //==============================================================
    // AUTOMATIC OPERATION
    //==============================================================
    automaticMode          : BOOL;    // EN: Automatic mode enable / PT: Habilita modo automático
    autoStopDelay          : TIME := T#1M;  // EN: Delay to stop pumps after machine stops / PT: Atraso para parar bombas após parada da máquina
END_VAR


VAR_OUTPUT
    //==============================================================
    // COMMANDS TO FIELD DEVICES
    //==============================================================
    pump1Run               : BOOL;    // EN: Run command for Pump 1 / PT: Comando de acionamento da Bomba 1
    pump2Run               : BOOL;    // EN: Run command for Pump 2 / PT: Comando de acionamento da Bomba 2

    //==============================================================
    // STATUS / FAULTS
    //==============================================================
    fault                  : BOOL;    // EN: General fault detected / PT: Falha geral detectada
    runningStatus          : BOOL;    // EN: TRUE if any pump is running / PT: TRUE se alguma bomba estiver ligada
    activePumpNumber       : INT;     // EN: 1 = Pump1, 2 = Pump2, 0 = None / PT: 1 = Bomba1, 2 = Bomba2, 0 = Nenhuma

    //==============================================================
    // STATE FEEDBACKS (FOR HMI DISPLAY)
    //==============================================================
    pump1State             : INT;     // EN: 0=Stopped, 1=Running, 3=Fault / PT: 0=Parada, 1=Rodando, 3 =Falha
    pump2State             : INT;     // EN: 0=Stopped, 1=Running, 3=Fault / PT: 0=Parada, 1=Rodando, 3 =Falha
	
    //==============================================================
    // FILTERED TEMPERATURE DISPLAY (FOR HMI)
    //==============================================================
    tankTemperatureFilteredDisplay    : REAL;  // EN: Filtered tank temperature [°C] / PT: Temperatura do tanque filtrada [°C]
    circuitTemperatureFilteredDisplay : REAL;  // EN: Filtered circuit temperature [°C] / PT: Temperatura do circuito filtrada [°C]
	
	
END_VAR


VAR
    //==============================================================
    // INTERNAL TIMERS / LOGIC FLAGS
    //==============================================================
    instTON_AutoStopDelay  : TON;     // EN: Timer to delay stop in automatic mode / PT: Temporizador de atraso de parada no modo automático
    autoRunRequest         : BOOL;    // EN: Internal flag for auto-start request / PT: Flag interna de solicitação de partida automática
    manualRunRequest       : BOOL;    // EN: Internal flag for manual start / PT: Flag interna de partida manual
    stopRequest            : BOOL;    // EN: Internal flag for stop request / PT: Flag interna de parada
    temperatureFault       : BOOL;    // EN: TRUE if abnormal temperature detected / PT: TRUE se temperatura anormal detectada

    //==============================================================
    // INTERNAL STATE CONTROL
    //==============================================================
    pump1StateInternal     : INT;     // EN: Internal logic state for Pump 1 / PT: Estado interno da Bomba 1
    pump2StateInternal     : INT;     // EN: Internal logic state for Pump 2 / PT: Estado interno da Bomba 2
    pump1RunCmd            : BOOL;    // EN: Command signal for Pump 1 / PT: Comando interno para Bomba 1
    pump2RunCmd            : BOOL;    // EN: Command signal for Pump 2 / PT: Comando interno para Bomba 2
	
    hmiAlarms                   : PaperMachine_TypeHmiAlarms; // Alarm structure / Estrutura de alarmes
	
    // EN: Delay to detect low pressure after pump start
    // PT: Atraso para detectar baixa pressão após partida da bomba
    tonLowPressure : TON;

    // EN: Delay to detect high pressure
    // PT: Atraso para detectar alta pressão
    tonHighPressure : TON;	
	
    //==============================================================
    // INTERNAL — FILTER INSTANCES
    //==============================================================
    instPT1_TankTemperatureDisplay    : FT_PT1;  // EN: Filter for tank temperature / PT: Filtro para temperatura do tanque
    instPT1_CircuitTemperatureDisplay : FT_PT1;  // EN: Filter for circuit temperature / PT: Filtro para temperatura do circuito
	
	startCmdOld : BOOL;  // EN: previous scan of startCmd / PT: estado anterior do startCmd
    rStartCmd   : BOOL;  // EN: rising edge of startCmd / PT: borda de subida do startCmd
    autoHoldAfterStop  : BOOL;   // EN: keep pump ON while delay is counting / PT: mantém bomba LIGADA enquanto o atraso conta
	
END_VAR

_PumpControl();
_FeedbackDisplay();
_alarmsDisplay();

METHOD _alarmsDisplay
VAR_INPUT
END_VAR
VAR


    // EN: TRUE when any pump is commanded to run
    // PT: TRUE quando qualquer bomba estiver comandada
    anyPumpEnabled : BOOL;
END_VAR


//==============================================================
// 1) ANY PUMP RUNNING?
//==============================================================
// EN: Consider enabled when we are actually commanding the pump outputs
// PT: Considera habilitada quando estamos realmente comandando as bombas
anyPumpEnabled := pump1Run OR pump2Run;


//==============================================================
// 2) LOW PRESSURE ALARM
//    EN: If any pump is enabled, we start a timer. If after the time
//        the minPressureFeedback is STILL FALSE, we raise the alarm.
//    PT: Se qualquer bomba estiver ligada, inicia o tempo. Se após o
//        tempo o minPressureFeedback continuar FALSE, disparamos o alarme.
//==============================================================
IF anyPumpEnabled THEN
    tonLowPressure(IN := NOT minPressureFeedback, PT := T#10S);
ELSE
    tonLowPressure(IN := FALSE);
END_IF;

IF tonLowPressure.Q THEN
    // EN: Low pressure after pump start → alarm
    // PT: Baixa pressão após partida da bomba → alarme
    hmiAlarms.lubricationMinPressureFaultAlarm := TRUE;

END_IF;


//==============================================================
// 3) HIGH / MAX PRESSURE ALARM
//    EN: We also wait a small time before setting max pressure alarm,
//        to avoid spikes at start.
//    PT: Também aguardamos um pequeno tempo antes de acusar alta pressão,
//        para evitar picos na partida.
//==============================================================
IF maxPressureFeedback THEN
    tonHighPressure(IN := TRUE, PT := T#30S);
ELSE
    tonHighPressure(IN := FALSE);
END_IF;

IF tonHighPressure.Q THEN
    hmiAlarms.lubricationMaxPressureFaultAlarm := TRUE;

END_IF;


//==============================================================
// TEMPERATURE ALARMS — LUBRIFICATION UNIT
// EN: Compares actual temperatures with configured max values
// PT: Compara as temperaturas medidas com os valores máximos configurados
//==============================================================

//------------------------------------
// 1) TANK TEMPERATURE ALARM
//------------------------------------
// EN: Alarm if tank temperature > tankMaxTemperature
// PT: Alarme se temperatura do tanque > tankMaxTemperature
IF tankTemperature > tankMaxTemperature THEN
    hmiAlarms.lubricationTankHighTemperatureAlarm := TRUE;     // EN: Tank temperature high / PT: Temperatura alta no tanque
END_IF;


//------------------------------------
// 2) CIRCUIT TEMPERATURE ALARM
//------------------------------------
// EN: Alarm if circuit temperature > circuitMaxTemperature
// PT: Alarme se temperatura do circuito > circuitMaxTemperature
IF circuitTemperature > circuitMaxTemperature THEN
    hmiAlarms.lubricationCircuitHighTemperatureAlarm := TRUE;  // EN: Circuit temperature high / PT: Temperatura alta no circuito
END_IF;


//==============================================================
// 4) PUMP FAULT MIRROR
//    EN: Just mirror field faults into HMI alarms
//    PT: Apenas reflete as falhas de campo para os alarmes da HMI
//==============================================================
hmiAlarms.lubricationPump1FaultAlarm := pump1Fault;   // EN: Pump 1 fault / PT: Falha bomba 1
hmiAlarms.lubricationPump2FaultAlarm := pump2Fault;   // EN: Pump 2 fault / PT: Falha bomba 2

fault  := hmiAlarms.lubricationMaxPressureFaultAlarm OR
		  hmiAlarms.lubricationMinPressureFaultAlarm OR 
		  (pump1Fault AND pump2Fault);
END_METHOD

METHOD _FeedbackDisplay
VAR_INPUT
END_VAR
//==============================================================
// TEMPERATURE FILTER LOGIC
// EN: Apply PT1 filtering for stable HMI visualization
// PT: Aplica filtro PT1 para visualização estável no supervisório
//==============================================================

instPT1_TankTemperatureDisplay(
    in  := tankTemperature,
    T   := T#10S,
    K   := 1.0,
    out => tankTemperatureFilteredDisplay
);

instPT1_CircuitTemperatureDisplay(
    IN := circuitTemperature,
    T   := T#10S,
    K   := 1.0,
    out => circuitTemperatureFilteredDisplay
);
END_METHOD

METHOD _PumpControl
VAR_INPUT
END_VAR


//------------------------------------
// 0) EDGE DETECTION FOR MANUAL START
//------------------------------------
// EN: manual start must work as a pulse → detect rising edge
// PT: partida manual deve funcionar por pulso → detecta borda de subida
rStartCmd   := (startCmd = TRUE) AND (startCmdOld = FALSE);
startCmdOld := startCmd;


//------------------------------------
// 1) BUILD RUN / STOP REQUESTS
//------------------------------------
// EN: manual run request is LATCHED until stopCmd (only in manual)
// PT: pedido de partida manual fica TRAVADO até stopCmd (apenas no manual)
IF rStartCmd THEN
    manualRunRequest := TRUE;
END_IF;

IF stopCmd AND (NOT automaticMode) THEN
    // EN: in manual we can stop
    // PT: em manual podemos parar
    manualRunRequest := FALSE;
END_IF;

// EN: defaults
// PT: valores padrão
autoRunRequest := FALSE;
stopRequest    := FALSE;

IF automaticMode THEN
    // EN: in automatic we do NOT allow stopCmd to stop pumps
    // PT: no automático NÃO deixamos o stopCmd desligar as bombas
    // (stopRequest stays FALSE)

    IF machineRunningFeedback THEN
        //======================================================
        // MACHINE RUNNING → RUN PUMP
        //======================================================
        autoRunRequest    := TRUE;
        autoHoldAfterStop := TRUE;                  // remember we were running
        instTON_AutoStopDelay(IN := FALSE);
    ELSE
        //======================================================
        // MACHINE STOPPED → START DELAY TO STOP
        //======================================================
        instTON_AutoStopDelay(IN := TRUE, PT := autoStopDelay);

        // EN: while delay is counting AND we were running before → keep running
        // PT: enquanto o atraso estiver contando E já estávamos rodando → mantém ligado
        IF (NOT instTON_AutoStopDelay.Q) AND autoHoldAfterStop THEN
            autoRunRequest := TRUE;
        ELSE
            autoRunRequest    := FALSE;
            autoHoldAfterStop := FALSE;             // release hold after delay
        END_IF;
    END_IF;

ELSE
    //----------------------------------------------------------
    // MANUAL MODE
    //----------------------------------------------------------
    stopRequest := FALSE;
    instTON_AutoStopDelay(IN := FALSE);
    autoHoldAfterStop := FALSE;
END_IF;


//------------------------------------
// 2) INITIAL SELECTION (OPERATOR)
//------------------------------------
// EN: FALSE → Pump 1, TRUE → Pump 2
// PT: FALSE → Bomba 1, TRUE → Bomba 2
IF pumpSelector = FALSE THEN
    activePumpNumber := 1;
ELSE
    activePumpNumber := 2;
END_IF;


//------------------------------------
// 3) MAIN START/STOP (single pump running)
//    EN: Run when (manualRunRequest OR autoRunRequest)
//    PT: Liga quando (manualRunRequest OU autoRunRequest)
//------------------------------------
IF (manualRunRequest OR autoRunRequest) THEN

    CASE activePumpNumber OF

        //======================================================
        // PUMP 1 SELECTED
        //======================================================
        1:
            IF NOT pump1Fault THEN
                // EN: selected pump OK → run pump 1
                // PT: bomba selecionada OK → liga bomba 1
                pump1RunCmd        := TRUE;
                pump1StateInternal := 1;   // running
                pump2RunCmd        := FALSE;
                IF NOT pump2Fault THEN
                    pump2StateInternal := 0;   // stopped
                END_IF;
            ELSE
                //==================================================
                // SELECTED PUMP FAULTED → TRY THE OTHER (AUTO ONLY)
                //==================================================
                // EN: Only in auto we are allowed to start the standby pump
                // PT: Somente no automático podemos acionar a bomba reserva
                IF NOT pump2Fault AND (autoRunRequest OR automaticMode) THEN
                    pump1RunCmd        := FALSE;
                    pump1StateInternal := 3;   // fault
                    pump2RunCmd        := TRUE;
                    pump2StateInternal := 1;   // running
                    activePumpNumber   := 2;   // update active pump for HMI
                ELSE
                    // EN: both faulted or we are in manual → stop outputs
                    // PT: ambas falhadas ou estamos no manual → desliga saídas
                    pump1RunCmd        := FALSE;
                    pump2RunCmd        := FALSE;
                    pump1StateInternal := 3;   // keep fault
                    IF pump2Fault THEN
                        pump2StateInternal := 3;
                    ELSE
                        pump2StateInternal := 0;
                    END_IF;
                END_IF;
            END_IF;

        //======================================================
        // PUMP 2 SELECTED
        //======================================================
        2:
            IF NOT pump2Fault THEN
                pump2RunCmd        := TRUE;
                pump2StateInternal := 1;   // running
                pump1RunCmd        := FALSE;
                IF NOT pump1Fault THEN
                    pump1StateInternal := 0;   // stopped
                END_IF;
            ELSE
                // selected pump (2) in fault → try pump 1 (auto only)
                IF NOT pump1Fault AND (autoRunRequest OR automaticMode) THEN
                    pump2RunCmd        := FALSE;
                    pump2StateInternal := 3;   // fault
                    pump1RunCmd        := TRUE;
                    pump1StateInternal := 1;   // running
                    activePumpNumber   := 1;   // update active pump for HMI
                ELSE
                    pump1RunCmd        := FALSE;
                    pump2RunCmd        := FALSE;
                    pump2StateInternal := 3;
                    IF pump1Fault THEN
                        pump1StateInternal := 3;
                    ELSE
                        pump1StateInternal := 0;
                    END_IF;
                END_IF;
            END_IF;

    ELSE
        //======================================================
        // INVALID SELECTION → STOP BOTH
        //======================================================
        pump1RunCmd        := FALSE;
        pump2RunCmd        := FALSE;
        IF pump1Fault THEN
            pump1StateInternal := 3;
        ELSE
            pump1StateInternal := 0;
        END_IF;
        IF pump2Fault THEN
            pump2StateInternal := 3;
        ELSE
            pump2StateInternal := 0;
        END_IF;
    END_CASE;

ELSE
    //==========================================================
    // NO RUN REQUEST → STOP BOTH (except keep fault states)
    // PT: Sem pedido de partida → desliga (mantendo falha)
    //==========================================================
    pump1RunCmd := FALSE;
    pump2RunCmd := FALSE;

    IF pump1Fault THEN
        pump1StateInternal := 3;
    ELSE
        pump1StateInternal := 0;
    END_IF;

    IF pump2Fault THEN
        pump2StateInternal := 3;
    ELSE
        pump2StateInternal := 0;
    END_IF;
END_IF;


//------------------------------------
// 4) MAP INTERNAL TO OUTPUTS
//------------------------------------
pump1Run   := pump1RunCmd;
pump2Run   := pump2RunCmd;

pump1State := pump1StateInternal;   // 0=Stopped,1=Running,3=Fault
pump2State := pump2StateInternal;   // 0=Stopped,1=Running,3=Fault


//------------------------------------
// 5) GLOBAL STATUS
//------------------------------------
runningStatus := pump1Run OR pump2Run;
END_METHOD

END_FUNCTION_BLOCK

// ---- Function Blocks/PaperMachine/Auxiliary/FB_SpeedDroopControl_1.TcPOU
FUNCTION_BLOCK FB_SpeedDroopControl_1
VAR_INPUT


	startGroup		: BOOL;
	groupFault		: BOOL;
	
	
	machineSpeedMPM	: REAL;
	
	machineMinSpeed	: REAL	:= 0.0;
	machineMaxSpeed	: REAL	:= 600.0;
	
	
	motorMaxSpeedMPM	: REAL := 600.0;
	
	
	speedAutoMan		: BOOL; //Speed selector (0 = Man / 1 = Auto)
	groupManualSpeedMPM	: REAL := 50.0;
	
	
	gearRatio : REAL := 1.0;
	
	
	recovery	: BOOL; //When pressed increase the group speed
	recoveryPct	: REAL;	//Paper recovery percentage this value is incremented to the speed setpoint	
	
	speedDifInc	: BOOL;
	speedDifDec	: BOOL;
	
	speedDifRate	: REAL := 0.1;
	speedDifLimLow	: REAL := -10.0;	
	speedDifLimHigh	: REAL := 10.0;

	
	rampRate	: REAL := 0.1;
	
	

END_VAR

VAR_OUTPUT
	
(*Slave setpoint variables*)
	driveSpeedRefPct  : REAL;		(*Speed reference to the drive*)
	driveSpeedRefPctRamp  : REAL;	(*Speed reference to the drive*)
	speedDifPct				: REAL;
	
	
	driveEnable		: BOOL;

END_VAR

VAR
	
	currentMachineSpeedPCT  : REAL;
	instTUNE2_SpeedDifGen	: TUNE2;
	instFB_Gen_SRamp	: FB_Gen_SRamp;

END_VAR

currentMachineSpeedPCT  := _Scale(machineSpeedMPM,0.0,machineMaxSpeed,0.0,100);


IF recovery THEN
	
	driveSpeedRefPct := (currentMachineSpeedPCT * gearRatio ) + speedDifPct;
	
ELSE
	
	driveSpeedRefPct := (currentMachineSpeedPCT * gearRatio ) + speedDifPct + recoveryPct; 

END_IF


_SpeedDifGenerator();
_RampGenerator();

METHOD _RampGenerator
VAR_INPUT
END_VAR
instFB_Gen_SRamp(
	X:= driveSpeedRefPct, 
	A_UP:= rampRate, 
	A_DN:= -rampRate, 
	VU_MAX:= 1.0, 
	VD_MAX:= -1.0, 
	LIMIT_HIGH:= 100.0, 
	LIMIT_LOW:= 0.0, 
	RST:= , 
	Y=> driveSpeedRefPctRamp, 
	V=> );
END_METHOD

METHOD PRIVATE _Scale : REAL
VAR_INPUT
	
	X : REAL;
	I_LO : REAL;
	I_HI : REAL;
	O_LO : REAL;
	O_HI : REAL;
	
END_VAR
IF I_LO = I_HI THEN
	_Scale := O_LO;
ELSE
	_Scale := (O_HI - O_LO) / (I_HI - I_LO) * (LIMIT(I_LO, X, I_HI) - I_LO) + O_LO;
END_IF;
END_METHOD

METHOD _SpeedDifGenerator
VAR_INPUT
END_VAR
instTUNE2_SpeedDifGen(
	SET:= , 
	SU:= speedDifInc, 
	SD:= speedDifDec, 
	FU:= , 
	FD:= , 
	RST:= , 
	SS:= speedDifRate, 
	FS:= speedDifRate, 
	Limit_L:= speedDifLimLow, 
	LIMIT_H:= speedDifLimHigh, 
	RST_val:= , 
	SET_val:= , 
	TR:= , 
	S1:= , 
	S2:= , 
	Y=> speedDifPct);
END_METHOD

END_FUNCTION_BLOCK

// ---- Function Blocks/PaperMachine/Auxiliary/FB_FormingBoardDriveControl.TcPOU
FUNCTION_BLOCK FB_FormingBoardDriveControl
VAR_INPUT
    // ── Group / Interlocks ───────────────────────────────────────────────────────
    startGroup                   : BOOL;   // Start command (Comando de partida)
    groupFault                   : BOOL;   // Fault present (Falha do grupo)
    groupMasterOperationEnabled  : BOOL;   // Master VFD "operation enabled"/running feedback
    groupSlaveOperationEnabled   : BOOL;   // Slave  VFD "operation enabled"/running feedback

    // ── Speed Setpoints ─────────────────────────────────────────────────────────
    groupAutoSpeedMPM        	 : REAL;   // Auto speed setpoint [m/min]
    groupMaxSpeed                : REAL := 600.0; // Max allowed line speed [m/min]

    // ── Auto / Manual ───────────────────────────────────────────────────────────
    groupSpeedAutoMan            : BOOL;   // 0=Manual / 1=Auto;
    groupManualSpeedMPM          : REAL := 50.0;  // Manual speed [m/min]

    // ── Feedbacks ───────────────────────────────────────────────────────────────
    masterTorqueFeedback         : REAL;   // [% or Nm]
    slaveTorqueFeedback          : REAL;   // [% or Nm]
    masterSpeedFeedback          : REAL;   // [m/min or %] — be consistent
    slaveSpeedFeedback           : REAL;   // [m/min or %] — be consistent

    // ── Ratio & Offsets ─────────────────────────────────────────────────────────
    gearRatio                    : REAL := 1.0;   // Slave/Master speed ratio
    slaveTorqueOfsset            : REAL := 0.0;          // (typo kept) torque trim [%/Nm]
    slaveSpeedOffset             : REAL := 10;          // Offset as % of master speed (+5 => +5%)
	
	// ── Torque control parameters ───────────────────────────────────────────────────
	torqueLimitMinPct    	: REAL := 5.0;   // Min torque [%]  (allow negative if regen, e.g. -100)
	torqueLimitMaxPct    	: REAL := 100.0; // Max torque [%]
	torqueDeadbandPct    	: REAL := 1.0;   // Below this |torque| => 0 (noise cleanup)
	torqueFilterTime		: TIME := T#20MS;

    // ── Dynamics (for ramp block) ───────────────────────────────────────────────
    rampRate                     : REAL := 0.01;  // Ref accel mag in %/s (A_UP=+rampRate, A_DN=-rampRate)
	
	// ── Speed diference limit ───────────────────────────────────────────────
	speedDiferenceLimit				: REAL := 20.0;
	
END_VAR

VAR_OUTPUT
	
	deviceState						: STRING;

    // ── Drive References (0..100%) ──────────────────────────────────────────────
    masterDriveSpeedRefPct       : REAL;   // Master reference [%]
    slaveDriveSpeedRefPct        : REAL;   // Slave  reference [%]
	nextGroupSpeedRefPct        	: REAL;   // Next group reference [%]


    slaveDriveTorqueLimit        : REAL;   // [% or Nm] (your logic)

    // ── Drive Commands ──────────────────────────────────────────────────────────
    masterDriveEnable            : BOOL;
    slaveDriveEnable             : BOOL;
    masterDriveReset             : BOOL;
    slaveDriveReset              : BOOL;
	currentSpeedDifence				: REAL;	

	
END_VAR

VAR
    // ── Internals ───────────────────────────────────────────────────────────────
    rampTargetPct                : REAL;   // 0..100% target into ramp
    instTUNE2_SpeedDifGen        : TUNE2;  // (reserved)
    instFB_Gen_SRamp             : FB_Gen_SRamp; // Your ramp FB

    // State machine
    state                        : INT;    // 0=IDLE,1=ENABLE,2=WAIT_EN,3=RAMP_EN,4=RUN,5=STOPPING,10=FAULT
    startGroupOld                : BOOL;
    rStart                       : BOOL;
    rStop                        : BOOL;

    // Timers
    instTONEnableWait            : TON;
    instTONStopWait              : TON;

    // Parameters for waits/thresholds
    enableTimeout                : TIME := T#5S;     // Wait for op-enable
    stopTimeout                  : TIME := T#8S;     // Max wait to speed≈0
    speedZeroThresholdPct        : REAL := 4.00;     // Consider stopped if |speed| ≤ this (same unit as refs)
    epsRefPct                    : REAL := 0.05;     // Small epsilon for ref≈0

    // Flags to ramp FB
    rampReset                    : BOOL;   // Resets ramp (sets Y/V to 0 in your FB)
	

	
	// ── Filter state ────────────────────────────────────────────────────────────────
	torqueFiltY          : REAL;          // last filtered torque
	torqueFiltInit       : BOOL;          // init flag (bumpless start)	
	instsFT_PT1TorqueFilter	: FT_PT1;	
		
	instTONSpeedDifDelay: TON;
END_VAR

// ─────────────────────────────────────────────────────────────
// 1) Group control state machine
//    - Handles START/STOP edges
//    - Manages ENABLE, STOPPING, and FAULT states
//    - Controls drive enable/reset commands
_GroupControl();

// ─────────────────────────────────────────────────────────────
// 2) Speed reference generation
//    - Scales Auto/Manual speed setpoints into 0..100%
//    - Applies acceleration/deceleration ramps
//    - Considers gear ratio and slave offset
//    - Clamps values to avoid saturation (>100%)
_ReferenceGenerator();

// ─────────────────────────────────────────────────────────────
// 3) Torque reference transfer
//    - Reads master torque feedback and applies PT1 filter
//    - Cleans noise with deadband and adds slave offset
//    - Limits the torque to configured min/max bounds
_TorqueReference();

// ─────────────────────────────────────────────────────────────
// 4) Speed difference monitoring
//    - Calculates absolute difference between master/slave speeds
//    - Updates currentSpeedDifence (for HMI/diagnostics)
//    - If difference exceeds limit, forces STOPPING state
_SpeedDifferenceCheck();

METHOD _GroupControl
VAR_INPUT
END_VAR
VAR
    speedsNearZero : BOOL;
    refNearZero    : BOOL;
    bothOpEnabled  : BOOL;
END_VAR
// ───────────────────────── Main execution ─────────────────────────────────────── // Edges 
rStart := startGroup AND NOT startGroupOld; rStop := NOT startGroup AND startGroupOld; startGroupOld := startGroup; 
// Feedback conditions (use your chosen unit for threshold; here using %) 

speedsNearZero := (ABS(masterSpeedFeedback) <= speedZeroThresholdPct) AND (ABS(slaveSpeedFeedback) <= speedZeroThresholdPct); 

// Also consider the reference itself near zero (in case feedback not available) 
refNearZero := ABS(masterDriveSpeedRefPct) <= epsRefPct; bothOpEnabled := groupMasterOperationEnabled AND groupSlaveOperationEnabled;



// ── State machine ───────────────────────────────────────────────────────────────
CASE state OF
    0: // IDLE
        deviceState := 'IDLE';
        rampReset := TRUE;                    // keep ramp reset at idle
        IF rStart AND NOT groupFault THEN
            state := 1;
        END_IF

    1: // ENABLE DRIVES
        deviceState := 'ENABLE_DRIVES';
        masterDriveEnable := TRUE;
        slaveDriveEnable  := TRUE;
        rampReset         := TRUE;            // still hold ramp reset

        instTONEnableWait(IN := TRUE, PT := enableTimeout);
        state := 2;

    2: // WAIT ENABLE FEEDBACK
        deviceState := 'WAIT_ENABLE_FEEDBACK';
        masterDriveEnable := TRUE;
        slaveDriveEnable  := TRUE;
        rampReset         := TRUE;

        instTONEnableWait(IN := TRUE, PT := enableTimeout);

        IF groupFault THEN
            instTONEnableWait(IN := FALSE);
            state := 10;
        ELSIF rStop THEN
            instTONEnableWait(IN := FALSE);
            state := 5;                       // go to controlled stop
        ELSIF bothOpEnabled THEN
            instTONEnableWait(IN := FALSE);
            state := 3;
        ELSIF instTONEnableWait.Q THEN
            instTONEnableWait(IN := FALSE);
            state := 10;                      // treat as fault (no enable feedback)
        END_IF

    3: // RAMP ENABLE (single-cycle gate)
        deviceState := 'RAMP_ENABLE';
        masterDriveEnable := TRUE;
        slaveDriveEnable  := TRUE;
        rampReset         := FALSE;           // release ramp now
        state := 4;

    4: // RUN
        IF groupSpeedAutoMan THEN
            deviceState := 'RUN (Auto)';
        ELSE
            deviceState := 'RUN (Manual)';
        END_IF;

        masterDriveEnable := TRUE;
        slaveDriveEnable  := TRUE;
        rampReset         := FALSE;

        IF groupFault THEN
            state := 10;
        ELSIF rStop THEN
            state := 5;
        END_IF

    5: // STOPPING (controlled)
        deviceState := 'STOPPING';
        masterDriveEnable := TRUE;            // keep enabled during decel
        slaveDriveEnable  := TRUE;
        rampReset         := FALSE;           // keep ramp active to ramp down

        // Start/keep stop wait
//        instTONStopWait(IN := TRUE, PT := stopTimeout);

        // Disable only when speed≈0 AND reference≈0 (backup)
        IF groupFault THEN
            instTONStopWait(IN := FALSE);
            state := 10;

        ELSIF speedsNearZero AND refNearZero THEN
            masterDriveEnable := FALSE;
            slaveDriveEnable  := FALSE;
            instTONStopWait(IN := FALSE);
            state := 0;

        ELSIF instTONStopWait.Q THEN
            masterDriveEnable := FALSE;
            slaveDriveEnable  := FALSE;
            instTONStopWait(IN := FALSE);
            state := 10;
        END_IF

    10: // FAULT
        deviceState := 'FAULT';
        rampReset         := TRUE;            // force ramp outputs to zero
        masterDriveEnable := FALSE;
        slaveDriveEnable  := FALSE;

        // Clear fault when fault disappears and start is low
        IF (NOT groupFault) AND (NOT startGroup) THEN
            state := 0;
        END_IF
END_CASE;
END_METHOD

METHOD _ReferenceGenerator
VAR
    headroomEpsPct      : REAL := 0.20;   // anti-chatter near 100%
    offsetPct           : REAL;
    denom               : REAL;
    maxMasterBySlave    : REAL;
    allowedCapPct       : REAL;
    currMasterPct       : REAL;
    currSlavePct        : REAL;
	targetPct: REAL;
	cmdSpeedMPM: REAL;
END_VAR
// 3) Scale to 0..100% for the drives (as you already have)

IF groupSpeedAutoMan THEN
	
	targetPct := _Scale(
		X    := groupAutoSpeedMPM,
		I_LO := 0.0,      I_HI := groupMaxSpeed,
		O_LO := 0.0,      O_HI := 100.0);
ELSE
	
	targetPct := _Scale(
		X    := groupManualSpeedMPM,
		I_LO := 0.0,      I_HI := groupMaxSpeed,
		O_LO := 0.0,      O_HI := 100.0);	

END_IF


// 4) During STOPPING/FAULT we want zero target; in STOPPING we still ramp down
IF state = 5 THEN
    rampTargetPct := 0.0;
ELSE
    rampTargetPct := targetPct;
END_IF;

// --- NEW: Pre-limit so SLAVE can’t exceed 100% for given gear + offset ---
offsetPct := slaveSpeedOffset * 0.01;
denom     := gearRatio + offsetPct;

// If denom <= 0, fall back to 100% (no additional cap required)
IF denom > 0.0 THEN
    maxMasterBySlave := 100.0 / denom;   // master % that makes slave hit 100%
ELSE
    maxMasterBySlave := 100.0;
END_IF;

// The cap the master target must obey (also respect master’s own 100%)
allowedCapPct := MIN(100.0, maxMasterBySlave);

// Apply cap to upward commands only (don’t block decel)
rampTargetPct := MIN(rampTargetPct, allowedCapPct);

// --- NEW: Freeze upward if currently at/near limit (anti-overrun using current refs) ---
currMasterPct := instFB_Gen_SRamp.Y;                          // current master ref (%)
currSlavePct  := LIMIT(0.0, currMasterPct * (gearRatio + offsetPct), 100.0);

IF (currMasterPct >= 100.0 - headroomEpsPct) OR
   (currSlavePct  >= 100.0 - headroomEpsPct) THEN
    // Prevent increasing the target above current value; allow decreases
    rampTargetPct := MIN(rampTargetPct, currMasterPct);
END_IF;

// 5) Ramp call (unchanged)
instFB_Gen_SRamp(
    X          := rampTargetPct,
    A_UP       := MAX(0.0, rampRate),
    A_DN       := -MAX(0.0, rampRate),
    VU_MAX     := 1000.0,
    VD_MAX     := -1000.0,
    LIMIT_HIGH := 100.0,
    LIMIT_LOW  := 3.5,
    RST        := rampReset);

// 6) Master reference = ramp Y but also respect the slave-driven cap
masterDriveSpeedRefPct := MIN(instFB_Gen_SRamp.Y, allowedCapPct);

// 7) Slave reference: gear + offset, then clamp 0..100
slaveDriveSpeedRefPct :=
    LIMIT(0.0, masterDriveSpeedRefPct * (gearRatio + offsetPct), 100.0);

// 8) Final safety clamp for master (already capped above, but keep it symmetrical)
masterDriveSpeedRefPct := LIMIT(0.0, masterDriveSpeedRefPct, 100.0);
nextGroupSpeedRefPct := masterDriveSpeedRefPct;
END_METHOD

METHOD PRIVATE _Scale : REAL
VAR_INPUT
	
	X : REAL;
	I_LO : REAL;
	I_HI : REAL;
	O_LO : REAL;
	O_HI : REAL;
	
END_VAR
IF I_LO = I_HI THEN
	_Scale := O_LO;
ELSE
	_Scale := (O_HI - O_LO) / (I_HI - I_LO) * (LIMIT(I_LO, X, I_HI) - I_LO) + O_LO;
END_IF;
END_METHOD

METHOD PRIVATE _SpeedDifferenceCheck
VAR
    diff : REAL;
END_VAR

// 1) Calcular diferença absoluta Master-Slave
diff := ABS(masterSpeedFeedback - slaveSpeedFeedback);
currentSpeedDifence := diff;

// 2) Se ultrapassar limite -> parar grupo
IF diff > speedDiferenceLimit THEN
    // Forçar parada de forma segura
	
	instTONSpeedDifDelay.IN := TRUE;
	instTONSpeedDifDelay.PT := T#5S;	
	
	IF instTONSpeedDifDelay.Q THEN

		state := 10;                  // vai para STOPPING (controlled stop)
		deviceState := 'FAULT: Speed difference exceeded';		
		
	END_IF
	
ELSE

	instTONSpeedDifDelay.IN := FALSE;
	
END_IF




instTONSpeedDifDelay();
END_METHOD

METHOD _TorqueReference
VAR
    rawTorque      : REAL;
    filtTorque     : REAL;
    torqueCmd      : REAL;
    limitedTorque  : REAL;
    alpha          : REAL;
    clamped        : BOOL;
	
END_VAR


// 1) Read master torque (keep units consistent with your limits)
rawTorque := masterTorqueFeedback;

// 2) Low-pass filter (OSCAT PT1)
instsFT_PT1TorqueFilter(
    in  := rawTorque,
    T   := torqueFilterTime,   // time constant in seconds (e.g., 0.25)
    K   := 0.8,                // unity gain
    out => filtTorque
);

// 3) Deadband cleanup
IF ABS(filtTorque) < torqueDeadbandPct THEN
    filtTorque := 0.0;
END_IF

// 4) Apply offset between master and slave
torqueCmd := filtTorque + slaveTorqueOfsset;

// 5) Clamp to limits
limitedTorque := LIMIT(torqueLimitMinPct, torqueCmd, torqueLimitMaxPct);
clamped       := (limitedTorque <> torqueCmd);

// 6) Output
slaveDriveTorqueLimit := limitedTorque;


//slaveDriveTorqueLimit := LIMIT(torqueLimitMinPct, masterTorqueFeedback, torqueLimitMaxPct);
END_METHOD

END_FUNCTION_BLOCK

// ---- Function Blocks/PaperMachine/DriveControl/FB_PressSectionDriveControl_V2.TcPOU
FUNCTION_BLOCK FB_PressSectionDriveControl_V2

VAR_INPUT

    //────────────────────────────────────────────
    // GROUP / INTERLOCKS
    //────────────────────────────────────────────
    startGroup              : BOOL; // Start command (pulse) / Comando de partida (pulso)
    stopGroup               : BOOL; // Stop command (level) / Comando de parada (nível)
    groupReset              : BOOL; // Fault reset / Reset de falhas do grupo
    groupFastStop           : BOOL;  // EN: Reset group faults / PT: Reset de falhas do grupo
	
    //────────────────────────────────────────────
    // AUXILIARY MOTORS — INDICATORS & COMMANDS
    //────────────────────────────────────────────
    grouSpeedDifIncCmd         : BOOL; // Lamp: offset increasing / Lâmpada: aumento de offset
    grouSpeedDifDecCmd         : BOOL; // Lamp: offset decreasing / Lâmpada: redução de offset
	
    //────────────────────────────────────────────
    // SPEED ADJUSTMENTS / OFFSET TUNING
    //────────────────────────────────────────────
    groupRecoverSpeedCmd    : BOOL; // Recover speed while TRUE / Recuperar velocidade enquanto TRUE


    //────────────────────────────────────────────
    // DRIVE STATUS INPUTS — PRESS SECTION (2 MOTORS)
    //────────────────────────────────────────────
    firstPressReady         : BOOL; // First press (MASTER) ready / Prensa 1 (mestre) pronto
    secondPressReady        : BOOL; // Second press (SLAVE) ready / Prensa 2 (escravo) pronto

    //────────────────────────────────────────────
    // SPEED SETPOINTS / MODE
    //────────────────────────────────────────────
    groupAutoSpeedMPM       : REAL; // Auto mode speed [m/min] / Velocidade em modo automático [m/min]
    groupManualSpeedMPM     : REAL := 50.0; // Manual mode speed / Velocidade em modo manual
    groupSpeedAutoMan       : BOOL; // Speed mode: 0=Manual, 1=Auto / Modo de velocidade: 0=Manual, 1=Automático

    //────────────────────────────────────────────
    // SPEED & TORQUE FEEDBACKS
    //────────────────────────────────────────────
    firstPressSpeedFeedback : REAL; // First press speed feedback / Velocidade medida da prensa 1
    firstPressTorqueFeedback: REAL; // First press torque feedback / Torque da prensa 1
    secondPressSpeedFeedback: REAL; // Second press speed feedback / Velocidade medida da prensa 2
    secondPressTorqueFeedback: REAL; // Second press torque feedback / Torque da prensa 2


    //──── Upper Felt 1 Stretcher ────
    upperFelt1StretcherCmdFwd     : BOOL; // Run forward / Comando para frente
    upperFelt1StretcherCmdRev     : BOOL; // Run reverse / Comando para trás
    upperFelt1StretcherFault      : BOOL; // Fault detected / Falha detectada
    upperFelt1StretcherLimitFwd   : BOOL; // End limit forward / Fim de curso frente
    upperFelt1StretcherLimitRev   : BOOL; // End limit reverse / Fim de curso trás

    //──── Upper Felt 2 Stretcher ────
    upperFelt2StretcherCmdFwd     : BOOL; // Run forward / Comando para frente
    upperFeltt2tretcherCmdRev     : BOOL; // Run reverse / Comando para trás (corrigir nome!)
    upperFeltS2tretcherFault      : BOOL; // Fault detected / Falha detectada
    upperFeltS2tretcherLimitFwd   : BOOL; // End limit forward / Fim de curso frente
    upperFeltS2tretcherLimitRev   : BOOL; // End limit reverse / Fim de curso trás

    //──── Lower Felt Stretcher ────
    lowerFeltStretcherCmdFwd      : BOOL;
    lowerFeltStretcherCmdRev      : BOOL;
    lowerFeltStretcherFault       : BOOL;
    lowerFeltStretcherLimitFwd    : BOOL;
    lowerFeltStretcherLimitRev    : BOOL;

    //──── Upper Infeed Roll ────
    upperInfeedRollCmdFwd         : BOOL;
    upperInfeedRollCmdRev         : BOOL;
    upperInfeedRollFault          : BOOL;
    upperInfeedRollLimitFwd       : BOOL;
    upperInfeedRollLimitRev       : BOOL;

    //──── Lower Infeed Roll ────
    lowerInfeedRollCmdFwd         : BOOL;
    lowerInfeedRollCmdRev         : BOOL;
    lowerInfeedRollFault          : BOOL;
    lowerInfeedRollLimitFwd       : BOOL;
    lowerInfeedRollLimitRev       : BOOL;

    //────────────────────────────────────────────
    // FELT EDGE / RUNNING SAFETY SENSORS
    //────────────────────────────────────────────
    pressSectionUpperFelt1OverrunSensorOperatorSide : BOOL; // Operator side / Lado operador
    pressSectionUpperFelt1OverrunSensorDriveSide    : BOOL; // Drive side / Lado comando

    pressSectionUpperFelt2OverrunSensorOperatorSide : BOOL;
    pressSectionUpperFelt2OverrunSensorDriveSide    : BOOL;

    pressSectionLowerFeltOverrunSensorOperatorSide  : BOOL;
    pressSectionLowerFeltOverrunSensorDriveSide     : BOOL;

	
	machineConfig			:  PaperMachine_TypeHmiConfig;
	
END_VAR



VAR_OUTPUT

    //────────────────────────────────────────────
    // STATE / DIAGNOSTICS
    //────────────────────────────────────────────
    deviceState                 : STRING; // Current state string / Estado atual em texto
    statusCode                  : INT;    // 0=Idle, 1=Starting, 2=Running, 3=Fault
    groupFault                  : BOOL;   // TRUE if any group fault active / Falha geral do grupo
	speedDif						: REAL;

    //────────────────────────────────────────────
    // SPEED REFERENCES (TO DRIVES) AND DISPLAY
    //────────────────────────────────────────────
    firstPressSpeedSetpointRPM  		: REAL; // Master speed reference [%] / Referência de velocidade mestre
    secondPressSpeedSetpointRPM 		: REAL; // Slave speed reference [%] / Referência de velocidade escravo 
	
	firstPressSpeedFeedbackRPM  		: REAL; // Master speed reference [%] / Referência de velocidade mestre
    secondPressSpeedFeedbackRPM 		: REAL; // Slave speed reference [%] / Referência de velocidade escravo 
	
	firstPressSpeedFeedbackMPM  		: REAL; // Master speed reference [%] / Referência de velocidade mestre
    secondPressSpeedFeedbackMPM 		: REAL; // Slave speed reference [%] / Referência de velocidade escravo 

	firstPressTorqueFeedbackPct  		: REAL; // Master speed reference [%] / Referência de velocidade mestre
    secondPressTorqueFeedbackPct 		: REAL; // Slave speed reference [%] / Referência de velocidade escravo 
	
	
	nextGroupSpeedRefMPM        : REAL; // Next group speed [m/min] / Velocidade do próximo grupo [m/min]

    //────────────────────────────────────────────
    // TORQUE REFERENCES / LIMITS (SLAVE)
    //────────────────────────────────────────────
    firstPressTorqueRefPct : REAL; // Torque setpoint for slave / Referência de torque escravo
//    secondPressTorqueRefPct : REAL; // Torque setpoint for slave / Referência de torque escravo

    //────────────────────────────────────────────
    // DRIVE COMMANDS (ENABLE / RESET)
    //────────────────────────────────────────────
    firstPressDriveEnable        : BOOL; // Enable master drive / Habilita drive mestre
    firstPressDriveReset         : BOOL; // Reset master drive fault / Reset falha drive mestre
    secondPressDriveEnable       : BOOL; // Enable slave drive / Habilita drive escravo
    secondPressDriveReset        : BOOL; // Reset slave drive fault / Reset falha drive escravo

    //────────────────────────────────────────────
    // STATUS CODES (PER DRIVE)
    //────────────────────────────────────────────
    firstPressStatusCode        : INT; // 0=Idle, 1=Start, 2=Run, 3=Fault / Código de status da prensa 1
    secondPressStatusCode       : INT; // Código de status da prensa 2

    //────────────────────────────────────────────
    // AUXILIARY MOTORS — DIRECT START OUTPUTS
    //────────────────────────────────────────────
    upperFelt1StretcherRunFwd   : BOOL; // Run forward / Rodar para frente
    upperFelt1StretcherRunRev   : BOOL; // Run reverse / Rodar para trás

